Yaskawa INFORM job: DEMO_ROOF_UPPER_0625_3PAINT_17.JBI

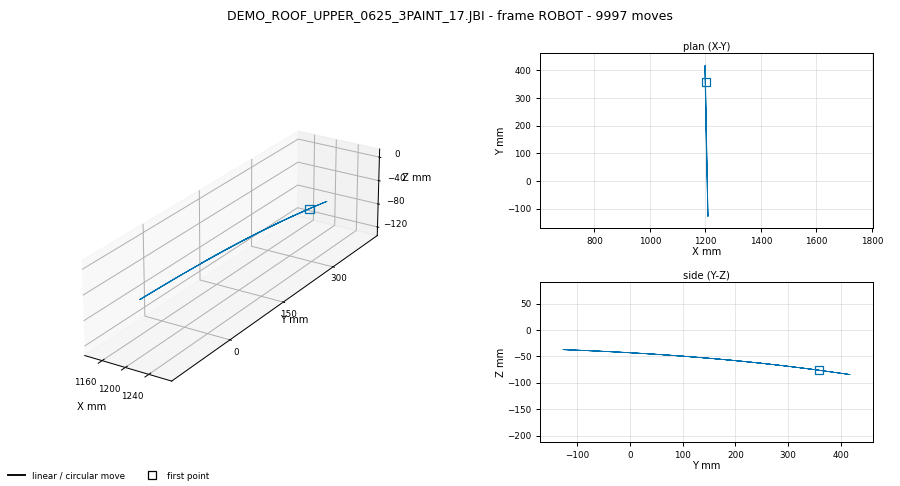
[picture p0: tool path of DEMO_ROOF_UPPER_0625_3PAINT_17.JBI in frame ROBOT, 9997 of 9997 moves have a stored position in this frame; points joined in program order, loops and branches not executed]
/JOB
//NAME DEMO_ROOF_UPPER_0625_3PAINT17
//POS
///NPOS 9997,0,0,0,0,0
///TOOL 0
///USER 0
///POSTYPE ROBOT
///RECTAN
///RCONF 1,0,0,0,0,0,0,0,0,0,0,0,0,0,0,0,0,0,0,0,0,0,0,0
C00000=1200.782,358.357,-76.024,-176.069,8.002,148.413
C00001=1200.786,358.109,-75.991,-176.071,7.999,148.412
C00002=1200.790,357.861,-75.958,-176.072,7.996,148.412
C00003=1200.794,357.613,-75.925,-176.074,7.993,148.412
C00004=1200.798,357.365,-75.891,-176.076,7.989,148.411
C00005=1200.802,357.118,-75.858,-176.078,7.987,148.411
C00006=1200.806,356.870,-75.825,-176.080,7.983,148.411
C00007=1200.811,356.622,-75.792,-176.082,7.980,148.410
C00008=1200.815,356.374,-75.759,-176.083,7.977,148.410
C00009=1200.818,356.127,-75.726,-176.085,7.974,148.410
C00010=1200.822,355.879,-75.693,-176.087,7.971,148.410
C00011=1200.826,355.632,-75.660,-176.089,7.967,148.409
C00012=1200.830,355.384,-75.627,-176.091,7.964,148.409
C00013=1200.835,355.136,-75.594,-176.093,7.962,148.409
C00014=1200.839,354.888,-75.560,-176.094,7.958,148.408
C00015=1200.843,354.641,-75.527,-176.097,7.955,148.408
C00016=1200.847,354.393,-75.494,-176.098,7.952,148.408
C00017=1200.851,354.145,-75.461,-176.101,7.949,148.408
C00018=1200.856,353.897,-75.429,-176.102,7.945,148.407
C00019=1200.860,353.649,-75.395,-176.104,7.943,148.407
C00020=1200.864,353.401,-75.362,-176.106,7.939,148.407
C00021=1200.867,353.154,-75.330,-176.108,7.936,148.406
C00022=1200.871,352.906,-75.297,-176.110,7.933,148.406
C00023=1200.876,352.658,-75.264,-176.112,7.930,148.406
C00024=1200.880,352.410,-75.231,-176.114,7.926,148.406
C00025=1200.884,352.162,-75.198,-176.116,7.924,148.406
C00026=1200.888,351.915,-75.165,-176.118,7.920,148.405
C00027=1200.892,351.667,-75.131,-176.120,7.917,148.405
C00028=1200.896,351.419,-75.100,-176.121,7.914,148.405
C00029=1200.900,351.171,-75.066,-176.124,7.911,148.405
C00030=1200.905,350.924,-75.034,-176.126,7.908,148.404
C00031=1200.909,350.676,-75.001,-176.128,7.905,148.404
C00032=1200.914,350.428,-74.968,-176.129,7.902,148.404
C00033=1200.917,350.181,-74.936,-176.132,7.898,148.404
C00034=1200.921,349.932,-74.903,-176.133,7.896,148.403
C00035=1200.926,349.685,-74.870,-176.135,7.892,148.403
C00036=1200.930,349.437,-74.837,-176.138,7.889,148.403
C00037=1200.934,349.189,-74.804,-176.139,7.887,148.403
C00038=1200.938,348.941,-74.772,-176.142,7.883,148.403
C00039=1200.942,348.693,-74.739,-176.144,7.880,148.402
C00040=1200.946,348.445,-74.706,-176.145,7.877,148.402
C00041=1200.951,348.198,-74.673,-176.147,7.874,148.402
C00042=1200.955,347.950,-74.642,-176.149,7.870,148.401
C00043=1200.959,347.702,-74.608,-176.152,7.867,148.401
C00044=1200.963,347.454,-74.576,-176.153,7.865,148.401
C00045=1200.967,347.206,-74.543,-176.156,7.861,148.401
C00046=1200.971,346.958,-74.511,-176.158,7.858,148.401
C00047=1200.975,346.710,-74.478,-176.159,7.855,148.400
C00048=1200.979,346.463,-74.446,-176.162,7.852,148.400
C00049=1200.984,346.215,-74.413,-176.164,7.849,148.400
C00050=1200.988,345.967,-74.381,-176.166,7.846,148.400
C00051=1200.991,345.720,-74.348,-176.168,7.843,148.400
C00052=1200.996,345.471,-74.316,-176.170,7.840,148.399
C00053=1201.000,345.223,-74.283,-176.172,7.837,148.399
C00054=1201.004,344.975,-74.251,-176.174,7.834,148.399
C00055=1201.008,344.728,-74.218,-176.176,7.830,148.399
C00056=1201.013,344.480,-74.186,-176.178,7.828,148.399
C00057=1201.017,344.232,-74.154,-176.180,7.825,148.398
C00058=1201.021,343.984,-74.121,-176.182,7.821,148.398
C00059=1201.025,343.736,-74.088,-176.184,7.819,148.398
C00060=1201.029,343.489,-74.057,-176.186,7.815,148.398
C00061=1201.034,343.241,-74.023,-176.189,7.812,148.398
C00062=1201.037,342.993,-73.992,-176.191,7.809,148.397
C00063=1201.042,342.745,-73.959,-176.193,7.806,148.397
C00064=1201.046,342.498,-73.927,-176.195,7.803,148.397
C00065=1201.050,342.249,-73.895,-176.197,7.800,148.397
C00066=1201.055,342.001,-73.862,-176.199,7.797,148.397
C00067=1201.058,341.754,-73.830,-176.201,7.794,148.396
C00068=1201.063,341.505,-73.797,-176.203,7.791,148.396
C00069=1201.067,341.258,-73.766,-176.205,7.788,148.396
C00070=1201.071,340.979,-73.729,-176.208,7.784,148.396
C00071=1201.076,340.702,-73.693,-176.210,7.781,148.396
C00072=1201.081,340.422,-73.657,-176.213,7.778,148.396
C00073=1201.086,340.144,-73.620,-176.215,7.774,148.395
C00074=1201.090,339.897,-73.589,-176.217,7.771,148.395
C00075=1201.094,339.649,-73.556,-176.219,7.769,148.395
C00076=1201.098,339.401,-73.524,-176.221,7.765,148.395
C00077=1201.101,339.153,-73.492,-176.224,7.762,148.395
C00078=1201.106,338.905,-73.460,-176.225,7.760,148.395
C00079=1201.110,338.657,-73.428,-176.227,7.756,148.394
C00080=1201.115,338.409,-73.396,-176.230,7.753,148.394
C00081=1201.119,338.161,-73.364,-176.232,7.750,148.394
C00082=1201.123,337.913,-73.332,-176.234,7.747,148.394
C00083=1201.127,337.665,-73.300,-176.236,7.744,148.394
C00084=1201.130,337.418,-73.267,-176.239,7.741,148.394
C00085=1201.136,337.170,-73.235,-176.241,7.738,148.394
C00086=1201.139,336.922,-73.203,-176.243,7.735,148.393
C00087=1201.144,336.673,-73.171,-176.245,7.732,148.393
C00088=1201.148,336.426,-73.140,-176.247,7.730,148.393
C00089=1201.152,336.178,-73.108,-176.249,7.726,148.393
C00090=1201.156,335.930,-73.075,-176.252,7.723,148.393
C00091=1201.160,335.682,-73.044,-176.254,7.720,148.392
C00092=1201.164,335.434,-73.012,-176.256,7.717,148.393
C00093=1201.169,335.186,-72.979,-176.258,7.714,148.392
C00094=1201.173,334.938,-72.949,-176.260,7.711,148.392
C00095=1201.177,334.690,-72.917,-176.263,7.708,148.392
C00096=1201.181,334.442,-72.884,-176.265,7.705,148.392
C00097=1201.186,334.194,-72.853,-176.267,7.702,148.392
C00098=1201.189,333.946,-72.821,-176.269,7.700,148.392
C00099=1201.194,333.699,-72.790,-176.271,7.696,148.392
C00100=1201.198,333.451,-72.757,-176.274,7.693,148.391
C00101=1201.202,333.203,-72.725,-176.276,7.690,148.391
C00102=1201.206,332.955,-72.694,-176.278,7.687,148.391
C00103=1201.210,332.707,-72.663,-176.281,7.684,148.391
C00104=1201.215,332.459,-72.631,-176.283,7.681,148.391
C00105=1201.219,332.211,-72.599,-176.285,7.679,148.391
C00106=1201.223,331.963,-72.567,-176.287,7.676,148.391
C00107=1201.227,331.716,-72.535,-176.289,7.672,148.391
C00108=1201.232,331.467,-72.504,-176.291,7.670,148.390
C00109=1201.236,331.219,-72.472,-176.294,7.667,148.390
C00110=1201.240,330.971,-72.440,-176.296,7.663,148.390
C00111=1201.244,330.724,-72.409,-176.298,7.661,148.390
C00112=1201.248,330.475,-72.378,-176.300,7.658,148.390
C00113=1201.252,330.227,-72.345,-176.303,7.655,148.390
C00114=1201.257,329.980,-72.314,-176.305,7.651,148.390
C00115=1201.261,329.731,-72.283,-176.307,7.649,148.390
C00116=1201.265,329.484,-72.251,-176.310,7.646,148.390
C00117=1201.269,329.235,-72.219,-176.312,7.643,148.389
C00118=1201.273,328.988,-72.189,-176.314,7.640,148.389
C00119=1201.278,328.739,-72.156,-176.316,7.637,148.389
C00120=1201.282,328.492,-72.125,-176.319,7.634,148.389
C00121=1201.286,328.243,-72.094,-176.321,7.631,148.389
C00122=1201.290,327.996,-72.062,-176.323,7.628,148.389
C00123=1201.294,327.747,-72.031,-176.325,7.625,148.389
C00124=1201.299,327.500,-72.000,-176.328,7.622,148.389
C00125=1201.302,327.252,-71.968,-176.330,7.620,148.389
C00126=1201.307,327.004,-71.937,-176.332,7.617,148.389
C00127=1201.311,326.756,-71.905,-176.335,7.613,148.388
C00128=1201.315,326.508,-71.874,-176.337,7.611,148.388
C00129=1201.319,326.260,-71.843,-176.339,7.608,148.388
C00130=1201.324,326.012,-71.812,-176.342,7.605,148.388
C00131=1201.327,325.764,-71.780,-176.343,7.602,148.388
C00132=1201.332,325.516,-71.749,-176.346,7.599,148.388
C00133=1201.336,325.268,-71.717,-176.348,7.596,148.388
C00134=1201.340,325.020,-71.687,-176.351,7.593,148.388
C00135=1201.344,324.772,-71.655,-176.353,7.591,148.388
C00136=1201.349,324.524,-71.624,-176.355,7.587,148.388
C00137=1201.353,324.275,-71.593,-176.358,7.584,148.388
C00138=1201.357,324.028,-71.561,-176.360,7.582,148.388
C00139=1201.361,323.779,-71.530,-176.362,7.579,148.388
C00140=1201.365,323.532,-71.499,-176.365,7.575,148.387
C00141=1201.370,323.284,-71.468,-176.367,7.573,148.387
C00142=1201.374,323.035,-71.437,-176.369,7.570,148.387
C00143=1201.378,322.788,-71.405,-176.372,7.567,148.387
C00144=1201.382,322.539,-71.374,-176.374,7.565,148.387
C00145=1201.387,322.291,-71.343,-176.376,7.561,148.387
C00146=1201.391,322.043,-71.312,-176.379,7.558,148.387
C00147=1201.395,321.795,-71.281,-176.381,7.556,148.387
C00148=1201.400,321.547,-71.250,-176.383,7.553,148.387
C00149=1201.404,321.299,-71.219,-176.386,7.550,148.387
C00150=1201.407,321.052,-71.188,-176.388,7.547,148.387
C00151=1201.412,320.804,-71.157,-176.390,7.544,148.387
C00152=1201.416,320.555,-71.126,-176.393,7.541,148.387
C00153=1201.421,320.307,-71.095,-176.395,7.538,148.387
C00154=1201.424,320.059,-71.064,-176.397,7.536,148.387
C00155=1201.429,319.811,-71.033,-176.400,7.533,148.387
C00156=1201.434,319.563,-71.002,-176.402,7.529,148.386
C00157=1201.437,319.315,-70.971,-176.404,7.527,148.386
C00158=1201.441,319.067,-70.941,-176.407,7.524,148.386
C00159=1201.446,318.819,-70.910,-176.410,7.521,148.386
C00160=1201.450,318.571,-70.878,-176.411,7.518,148.386
C00161=1201.454,318.323,-70.847,-176.414,7.515,148.386
C00162=1201.458,318.075,-70.817,-176.417,7.512,148.386
C00163=1201.462,317.827,-70.786,-176.418,7.510,148.386
C00164=1201.467,317.579,-70.755,-176.421,7.507,148.386
C00165=1201.471,317.331,-70.725,-176.424,7.504,148.386
C00166=1201.475,317.082,-70.694,-176.425,7.501,148.386
C00167=1201.479,316.834,-70.663,-176.428,7.498,148.386
C00168=1201.484,316.586,-70.632,-176.431,7.495,148.386
C00169=1201.488,316.338,-70.601,-176.433,7.492,148.386
C00170=1201.492,316.090,-70.571,-176.435,7.490,148.386
C00171=1201.497,315.842,-70.540,-176.438,7.487,148.386
C00172=1201.501,315.594,-70.510,-176.440,7.484,148.386
C00173=1201.505,315.345,-70.478,-176.443,7.482,148.386
C00174=1201.510,315.070,-70.444,-176.445,7.478,148.386
C00175=1201.515,314.793,-70.411,-176.447,7.475,148.386
C00176=1201.518,314.517,-70.377,-176.450,7.472,148.386
C00177=1201.523,314.241,-70.342,-176.453,7.468,148.386
C00178=1201.528,313.993,-70.312,-176.456,7.466,148.386
C00179=1201.533,313.745,-70.282,-176.458,7.463,148.385
C00180=1201.536,313.496,-70.251,-176.460,7.460,148.385
C00181=1201.541,313.248,-70.220,-176.463,7.458,148.385
C00182=1201.545,313.000,-70.189,-176.465,7.454,148.385
C00183=1201.549,312.753,-70.159,-176.468,7.451,148.386
C00184=1201.554,312.505,-70.129,-176.470,7.449,148.385
C00185=1201.558,312.256,-70.097,-176.472,7.446,148.385
C00186=1201.562,312.008,-70.068,-176.475,7.443,148.385
C00187=1201.567,311.760,-70.037,-176.477,7.441,148.385
C00188=1201.570,311.512,-70.007,-176.480,7.438,148.385
C00189=1201.574,311.264,-69.976,-176.482,7.434,148.385
C00190=1201.579,311.015,-69.946,-176.484,7.432,148.385
C00191=1201.583,310.767,-69.916,-176.487,7.429,148.385
C00192=1201.588,310.520,-69.885,-176.490,7.426,148.385
C00193=1201.592,310.272,-69.855,-176.492,7.424,148.385
C00194=1201.597,310.023,-69.825,-176.494,7.421,148.385
C00195=1201.600,309.775,-69.794,-176.497,7.418,148.385
C00196=1201.605,309.527,-69.763,-176.499,7.415,148.385
C00197=1201.609,309.279,-69.734,-176.501,7.412,148.385
C00198=1201.613,309.031,-69.703,-176.504,7.410,148.385
C00199=1201.617,308.783,-69.673,-176.506,7.407,148.385
C00200=1201.622,308.535,-69.643,-176.509,7.404,148.385
C00201=1201.626,308.287,-69.613,-176.511,7.402,148.385
C00202=1201.630,308.038,-69.582,-176.513,7.399,148.385
C00203=1201.634,307.790,-69.552,-176.516,7.396,148.385
C00204=1201.639,307.542,-69.521,-176.518,7.393,148.385
C00205=1201.643,307.294,-69.492,-176.521,7.390,148.385
C00206=1201.647,307.046,-69.462,-176.523,7.387,148.385
C00207=1201.652,306.798,-69.432,-176.526,7.385,148.385
C00208=1201.656,306.550,-69.402,-176.528,7.382,148.385
C00209=1201.661,306.301,-69.372,-176.531,7.379,148.385
C00210=1201.664,306.054,-69.341,-176.533,7.377,148.385
C00211=1201.669,305.804,-69.311,-176.535,7.374,148.385
C00212=1201.673,305.557,-69.281,-176.538,7.371,148.385
C00213=1201.677,305.308,-69.251,-176.540,7.368,148.385
C00214=1201.681,305.060,-69.221,-176.543,7.365,148.385
C00215=1201.686,304.812,-69.191,-176.545,7.363,148.385
C00216=1201.689,304.565,-69.161,-176.548,7.360,148.385
C00217=1201.694,304.316,-69.131,-176.550,7.357,148.385
C00218=1201.699,304.068,-69.101,-176.553,7.355,148.385
C00219=1201.703,303.820,-69.071,-176.555,7.352,148.385
C00220=1201.707,303.572,-69.041,-176.558,7.349,148.385
C00221=1201.711,303.324,-69.011,-176.560,7.347,148.386
C00222=1201.716,303.075,-68.981,-176.563,7.344,148.386
C00223=1201.720,302.827,-68.952,-176.565,7.341,148.386
C00224=1201.724,302.579,-68.921,-176.567,7.338,148.385
C00225=1201.728,302.331,-68.892,-176.570,7.335,148.385
C00226=1201.733,302.083,-68.862,-176.572,7.333,148.385
C00227=1201.738,301.834,-68.832,-176.575,7.330,148.385
C00228=1201.741,301.587,-68.802,-176.577,7.327,148.385
C00229=1201.746,301.338,-68.773,-176.579,7.325,148.386
C00230=1201.750,301.090,-68.743,-176.582,7.322,148.386
C00231=1201.754,300.842,-68.713,-176.584,7.319,148.386
C00232=1201.759,300.594,-68.683,-176.587,7.316,148.386
C00233=1201.763,300.346,-68.654,-176.590,7.313,148.386
C00234=1201.768,300.097,-68.624,-176.592,7.311,148.386
C00235=1201.772,299.849,-68.594,-176.594,7.308,148.386
C00236=1201.776,299.601,-68.564,-176.597,7.305,148.386
C00237=1201.780,299.353,-68.535,-176.599,7.303,148.386
C00238=1201.784,299.105,-68.505,-176.602,7.300,148.386
C00239=1201.789,298.856,-68.475,-176.604,7.298,148.386
C00240=1201.793,298.608,-68.446,-176.607,7.295,148.386
C00241=1201.797,298.359,-68.416,-176.610,7.292,148.386
C00242=1201.802,298.111,-68.387,-176.612,7.290,148.386
C00243=1201.805,297.864,-68.357,-176.614,7.287,148.386
C00244=1201.810,297.615,-68.327,-176.616,7.284,148.386
C00245=1201.814,297.367,-68.298,-176.619,7.281,148.386
C00246=1201.819,297.118,-68.268,-176.622,7.278,148.386
C00247=1201.823,296.870,-68.238,-176.624,7.276,148.386
C00248=1201.827,296.622,-68.209,-176.627,7.273,148.386
C00249=1201.832,296.374,-68.180,-176.629,7.271,148.386
C00250=1201.836,296.126,-68.150,-176.632,7.268,148.386
C00251=1201.840,295.878,-68.121,-176.635,7.265,148.387
C00252=1201.844,295.630,-68.091,-176.637,7.263,148.387
C00253=1201.849,295.381,-68.062,-176.640,7.260,148.387
C00254=1201.853,295.133,-68.032,-176.642,7.258,148.387
C00255=1201.857,294.885,-68.003,-176.644,7.255,148.387
C00256=1201.861,294.636,-67.973,-176.647,7.252,148.387
C00257=1201.865,294.388,-67.944,-176.649,7.250,148.387
C00258=1201.870,294.141,-67.915,-176.652,7.247,148.387
C00259=1201.875,293.892,-67.886,-176.654,7.244,148.387
C00260=1201.879,293.643,-67.857,-176.657,7.241,148.387
C00261=1201.883,293.395,-67.827,-176.659,7.238,148.387
C00262=1201.887,293.147,-67.798,-176.662,7.236,148.387
C00263=1201.891,292.899,-67.768,-176.664,7.233,148.387
C00264=1201.895,292.650,-67.739,-176.666,7.231,148.387
C00265=1201.900,292.403,-67.710,-176.670,7.228,148.387
C00266=1201.905,292.154,-67.681,-176.672,7.226,148.387
C00267=1201.909,291.906,-67.652,-176.674,7.223,148.387
C00268=1201.913,291.657,-67.622,-176.677,7.220,148.387
C00269=1201.917,291.409,-67.593,-176.679,7.218,148.387
C00270=1201.922,291.162,-67.564,-176.682,7.215,148.388
C00271=1201.927,290.913,-67.535,-176.684,7.213,148.388
C00272=1201.931,290.664,-67.505,-176.687,7.210,148.388
C00273=1201.935,290.416,-67.476,-176.689,7.207,148.388
C00274=1201.939,290.168,-67.448,-176.692,7.204,148.388
C00275=1201.943,289.920,-67.419,-176.695,7.202,148.388
C00276=1201.948,289.672,-67.389,-176.697,7.199,148.388
C00277=1201.952,289.423,-67.360,-176.700,7.196,148.388
C00278=1201.957,289.149,-67.328,-176.702,7.193,148.388
C00279=1201.962,288.874,-67.296,-176.705,7.190,148.388
C00280=1201.966,288.599,-67.264,-176.708,7.189,148.388
C00281=1201.971,288.326,-67.232,-176.710,7.186,148.388
C00282=1201.976,288.077,-67.203,-176.713,7.183,148.388
C00283=1201.980,287.829,-67.174,-176.715,7.180,148.388
C00284=1201.984,287.581,-67.144,-176.718,7.177,148.388
C00285=1201.988,287.332,-67.116,-176.720,7.174,148.389
C00286=1201.993,287.085,-67.087,-176.723,7.172,148.389
C00287=1201.997,286.836,-67.058,-176.726,7.169,148.389
C00288=1202.002,286.588,-67.029,-176.728,7.167,148.389
C00289=1202.005,286.339,-67.001,-176.731,7.164,148.389
C00290=1202.010,286.091,-66.972,-176.733,7.162,148.389
C00291=1202.015,285.843,-66.943,-176.735,7.159,148.389
C00292=1202.019,285.594,-66.913,-176.738,7.157,148.389
C00293=1202.023,285.346,-66.886,-176.741,7.154,148.389
C00294=1202.027,285.098,-66.856,-176.743,7.152,148.389
C00295=1202.032,284.849,-66.827,-176.746,7.149,148.389
C00296=1202.037,284.602,-66.798,-176.748,7.146,148.389
C00297=1202.040,284.353,-66.770,-176.751,7.144,148.390
C00298=1202.044,284.105,-66.741,-176.754,7.141,148.390
C00299=1202.050,283.857,-66.712,-176.756,7.139,148.390
C00300=1202.053,283.608,-66.684,-176.758,7.136,148.390
C00301=1202.057,283.360,-66.655,-176.761,7.134,148.390
C00302=1202.063,283.112,-66.626,-176.764,7.131,148.390
C00303=1202.066,282.863,-66.598,-176.766,7.129,148.390
C00304=1202.070,282.615,-66.569,-176.769,7.126,148.390
C00305=1202.076,282.367,-66.540,-176.771,7.124,148.390
C00306=1202.079,282.118,-66.512,-176.773,7.121,148.390
C00307=1202.084,281.870,-66.483,-176.776,7.119,148.391
C00308=1202.089,281.622,-66.455,-176.779,7.116,148.391
C00309=1202.092,281.373,-66.426,-176.781,7.113,148.391
C00310=1202.097,281.125,-66.397,-176.784,7.110,148.391
C00311=1202.102,280.877,-66.369,-176.786,7.108,148.391
C00312=1202.105,280.628,-66.340,-176.789,7.106,148.391
C00313=1202.110,280.380,-66.312,-176.791,7.103,148.391
C00314=1202.114,280.131,-66.284,-176.794,7.100,148.391
C00315=1202.119,279.884,-66.255,-176.796,7.098,148.391
C00316=1202.123,279.635,-66.227,-176.799,7.096,148.392
C00317=1202.127,279.386,-66.198,-176.801,7.093,148.392
C00318=1202.132,279.138,-66.170,-176.804,7.090,148.392
C00319=1202.136,278.889,-66.141,-176.806,7.088,148.392
C00320=1202.140,278.642,-66.113,-176.809,7.085,148.392
C00321=1202.145,278.393,-66.084,-176.811,7.083,148.392
C00322=1202.149,278.145,-66.056,-176.814,7.080,148.392
C00323=1202.153,277.897,-66.028,-176.816,7.078,148.392
C00324=1202.157,277.648,-66.000,-176.819,7.075,148.392
C00325=1202.162,277.400,-65.971,-176.821,7.073,148.393
C00326=1202.166,277.151,-65.943,-176.824,7.070,148.393
C00327=1202.171,276.903,-65.915,-176.826,7.068,148.393
C00328=1202.175,276.654,-65.886,-176.830,7.065,148.393
C00329=1202.180,276.406,-65.858,-176.832,7.063,148.393
C00330=1202.184,276.158,-65.830,-176.834,7.060,148.393
C00331=1202.189,275.909,-65.802,-176.837,7.058,148.393
C00332=1202.193,275.661,-65.773,-176.840,7.055,148.393
C00333=1202.198,275.413,-65.745,-176.842,7.053,148.393
C00334=1202.201,275.164,-65.717,-176.845,7.050,148.393
C00335=1202.206,274.916,-65.689,-176.847,7.048,148.394
C00336=1202.210,274.667,-65.660,-176.850,7.045,148.394
C00337=1202.215,274.419,-65.633,-176.852,7.043,148.394
C00338=1202.219,274.171,-65.604,-176.855,7.041,148.394
C00339=1202.223,273.923,-65.576,-176.857,7.038,148.394
C00340=1202.227,273.674,-65.548,-176.859,7.036,148.394
C00341=1202.232,273.426,-65.520,-176.862,7.033,148.394
C00342=1202.236,273.177,-65.491,-176.865,7.031,148.395
C00343=1202.240,272.930,-65.464,-176.867,7.028,148.395
C00344=1202.246,272.681,-65.436,-176.870,7.026,148.395
C00345=1202.249,272.432,-65.408,-176.873,7.023,148.395
C00346=1202.254,272.184,-65.380,-176.875,7.021,148.395
C00347=1202.258,271.935,-65.351,-176.878,7.018,148.395
C00348=1202.263,271.687,-65.324,-176.880,7.016,148.395
C00349=1202.266,271.439,-65.295,-176.882,7.014,148.395
C00350=1202.271,271.190,-65.268,-176.885,7.011,148.395
C00351=1202.276,270.942,-65.240,-176.888,7.009,148.396
C00352=1202.280,270.694,-65.212,-176.890,7.006,148.396
C00353=1202.284,270.446,-65.184,-176.893,7.004,148.396
C00354=1202.289,270.196,-65.156,-176.896,7.001,148.396
C00355=1202.293,269.948,-65.128,-176.898,6.999,148.396
C00356=1202.297,269.700,-65.100,-176.901,6.996,148.396
C00357=1202.302,269.451,-65.073,-176.903,6.994,148.397
C00358=1202.307,269.203,-65.045,-176.905,6.992,148.397
C00359=1202.311,268.955,-65.017,-176.908,6.989,148.397
C00360=1202.315,268.706,-64.990,-176.911,6.987,148.397
C00361=1202.320,268.458,-64.962,-176.913,6.984,148.397
C00362=1202.323,268.210,-64.934,-176.915,6.982,148.397
C00363=1202.329,267.961,-64.906,-176.919,6.979,148.397
C00364=1202.333,267.713,-64.878,-176.921,6.977,148.397
C00365=1202.337,267.464,-64.850,-176.923,6.975,148.398
C00366=1202.342,267.216,-64.823,-176.926,6.972,148.398
C00367=1202.346,266.968,-64.795,-176.928,6.970,148.398
C00368=1202.350,266.719,-64.768,-176.931,6.967,148.398
C00369=1202.355,266.471,-64.739,-176.934,6.965,148.398
C00370=1202.360,266.222,-64.712,-176.936,6.962,148.398
C00371=1202.363,265.974,-64.684,-176.939,6.960,148.399
C00372=1202.368,265.725,-64.657,-176.941,6.958,148.399
C00373=1202.372,265.477,-64.629,-176.944,6.955,148.399
C00374=1202.377,265.228,-64.602,-176.946,6.953,148.399
C00375=1202.381,264.980,-64.574,-176.949,6.950,148.399
C00376=1202.386,264.732,-64.547,-176.952,6.948,148.399
C00377=1202.389,264.483,-64.519,-176.954,6.946,148.399
C00378=1202.394,264.235,-64.492,-176.957,6.943,148.399
C00379=1202.399,263.986,-64.464,-176.959,6.941,148.400
C00380=1202.404,263.738,-64.436,-176.962,6.938,148.400
C00381=1202.407,263.489,-64.408,-176.964,6.936,148.400
C00382=1202.412,263.217,-64.379,-176.967,6.933,148.400
C00383=1202.418,262.944,-64.349,-176.970,6.932,148.400
C00384=1202.422,262.670,-64.318,-176.973,6.929,148.400
C00385=1202.427,262.398,-64.289,-176.976,6.926,148.401
C00386=1202.431,262.150,-64.261,-176.978,6.924,148.401
C00387=1202.436,261.902,-64.234,-176.981,6.921,148.401
C00388=1202.440,261.652,-64.206,-176.983,6.919,148.401
C00389=1202.444,261.405,-64.179,-176.985,6.917,148.401
C00390=1202.449,261.156,-64.152,-176.989,6.914,148.402
C00391=1202.453,260.908,-64.124,-176.991,6.912,148.402
C00392=1202.458,260.658,-64.097,-176.993,6.910,148.402
C00393=1202.462,260.411,-64.069,-176.996,6.907,148.402
C00394=1202.467,260.162,-64.042,-176.999,6.905,148.402
C00395=1202.471,259.914,-64.015,-177.001,6.902,148.402
C00396=1202.476,259.665,-63.988,-177.003,6.900,148.402
C00397=1202.480,259.416,-63.960,-177.006,6.898,148.403
C00398=1202.484,259.168,-63.933,-177.009,6.895,148.403
C00399=1202.488,258.920,-63.906,-177.011,6.893,148.403
C00400=1202.493,258.671,-63.879,-177.014,6.891,148.403
C00401=1202.497,258.423,-63.852,-177.017,6.888,148.403
C00402=1202.501,258.174,-63.824,-177.019,6.886,148.403
C00403=1202.506,257.926,-63.797,-177.022,6.884,148.404
C00404=1202.511,257.677,-63.770,-177.024,6.881,148.404
C00405=1202.515,257.429,-63.743,-177.027,6.879,148.404
C00406=1202.520,257.180,-63.716,-177.029,6.877,148.404
C00407=1202.524,256.932,-63.689,-177.032,6.874,148.404
C00408=1202.528,256.684,-63.662,-177.034,6.872,148.405
C00409=1202.532,256.434,-63.635,-177.037,6.869,148.405
C00410=1202.537,256.186,-63.608,-177.040,6.867,148.405
C00411=1202.542,255.937,-63.581,-177.042,6.865,148.405
C00412=1202.546,255.689,-63.554,-177.045,6.863,148.405
C00413=1202.550,255.441,-63.527,-177.047,6.860,148.405
C00414=1202.555,255.192,-63.500,-177.050,6.859,148.406
C00415=1202.560,254.944,-63.473,-177.052,6.856,148.406
C00416=1202.564,254.695,-63.446,-177.055,6.854,148.406
C00417=1202.568,254.446,-63.419,-177.057,6.852,148.406
C00418=1202.572,254.198,-63.392,-177.060,6.849,148.406
C00419=1202.577,253.949,-63.365,-177.063,6.847,148.407
C00420=1202.582,253.701,-63.338,-177.065,6.845,148.407
C00421=1202.586,253.453,-63.312,-177.067,6.843,148.407
C00422=1202.590,253.204,-63.285,-177.071,6.840,148.407
C00423=1202.595,252.956,-63.257,-177.073,6.838,148.407
C00424=1202.599,252.707,-63.231,-177.075,6.836,148.408
C00425=1202.603,252.459,-63.204,-177.078,6.833,148.408
C00426=1202.608,252.211,-63.177,-177.081,6.831,148.408
C00427=1202.613,251.962,-63.150,-177.083,6.829,148.408
C00428=1202.617,251.713,-63.124,-177.086,6.826,148.408
C00429=1202.622,251.465,-63.097,-177.088,6.824,148.408
C00430=1202.626,251.216,-63.070,-177.091,6.822,148.409
C00431=1202.630,250.968,-63.043,-177.093,6.819,148.409
C00432=1202.634,250.719,-63.016,-177.096,6.817,148.409
C00433=1202.638,250.471,-62.990,-177.098,6.815,148.409
C00434=1202.643,250.222,-62.963,-177.101,6.813,148.409
C00435=1202.648,249.973,-62.936,-177.104,6.810,148.410
C00436=1202.652,249.725,-62.910,-177.106,6.808,148.410
C00437=1202.656,249.476,-62.883,-177.108,6.806,148.410
C00438=1202.661,249.227,-62.856,-177.112,6.804,148.410
C00439=1202.665,248.979,-62.830,-177.114,6.801,148.410
C00440=1202.670,248.731,-62.803,-177.116,6.800,148.411
C00441=1202.674,248.482,-62.777,-177.119,6.797,148.411
C00442=1202.679,248.233,-62.750,-177.122,6.795,148.411
C00443=1202.683,247.985,-62.724,-177.124,6.793,148.411
C00444=1202.688,247.736,-62.697,-177.126,6.791,148.411
C00445=1202.693,247.488,-62.670,-177.130,6.788,148.412
C00446=1202.697,247.240,-62.644,-177.132,6.786,148.412
C00447=1202.702,246.991,-62.618,-177.134,6.784,148.412
C00448=1202.706,246.743,-62.591,-177.137,6.781,148.412
C00449=1202.710,246.494,-62.564,-177.140,6.779,148.412
C00450=1202.715,246.245,-62.538,-177.142,6.777,148.413
C00451=1202.719,245.997,-62.511,-177.145,6.775,148.413
C00452=1202.723,245.748,-62.486,-177.148,6.772,148.413
C00453=1202.728,245.500,-62.458,-177.150,6.770,148.413
C00454=1202.732,245.251,-62.433,-177.152,6.768,148.414
C00455=1202.737,245.002,-62.406,-177.155,6.766,148.414
C00456=1202.741,244.753,-62.380,-177.158,6.764,148.414
C00457=1202.745,244.505,-62.353,-177.160,6.761,148.414
C00458=1202.750,244.257,-62.326,-177.163,6.760,148.414
C00459=1202.754,244.008,-62.301,-177.165,6.758,148.415
C00460=1202.760,243.760,-62.275,-177.168,6.755,148.415
C00461=1202.764,243.511,-62.248,-177.171,6.753,148.415
C00462=1202.768,243.262,-62.222,-177.173,6.751,148.415
C00463=1202.772,243.014,-62.195,-177.175,6.749,148.415
C00464=1202.777,242.765,-62.170,-177.178,6.746,148.415
C00465=1202.781,242.517,-62.143,-177.181,6.744,148.416
C00466=1202.786,242.268,-62.117,-177.183,6.742,148.416
C00467=1202.790,242.019,-62.090,-177.185,6.740,148.416
C00468=1202.794,241.771,-62.064,-177.189,6.737,148.416
C00469=1202.799,241.523,-62.039,-177.191,6.735,148.417
C00470=1202.804,241.274,-62.012,-177.193,6.733,148.417
C00471=1202.808,241.025,-61.986,-177.196,6.731,148.417
C00472=1202.812,240.776,-61.960,-177.199,6.728,148.417
C00473=1202.817,240.528,-61.933,-177.201,6.727,148.418
C00474=1202.821,240.279,-61.907,-177.204,6.724,148.418
C00475=1202.826,240.031,-61.882,-177.206,6.723,148.418
C00476=1202.831,239.783,-61.855,-177.209,6.720,148.418
C00477=1202.835,239.534,-61.829,-177.212,6.718,148.418
C00478=1202.839,239.285,-61.803,-177.214,6.716,148.419
C00479=1202.844,239.036,-61.777,-177.217,6.714,148.419
C00480=1202.849,238.788,-61.751,-177.219,6.712,148.419
C00481=1202.853,238.540,-61.725,-177.222,6.709,148.419
C00482=1202.857,238.291,-61.699,-177.224,6.707,148.419
C00483=1202.862,238.042,-61.673,-177.227,6.705,148.420
C00484=1202.866,237.793,-61.647,-177.230,6.703,148.420
C00485=1202.871,237.545,-61.621,-177.232,6.700,148.420
C00486=1202.875,237.273,-61.593,-177.235,6.699,148.421
C00487=1202.880,237.002,-61.565,-177.238,6.696,148.421
C00488=1202.886,236.731,-61.536,-177.241,6.694,148.421
C00489=1202.891,236.459,-61.508,-177.244,6.691,148.421
C00490=1202.895,236.210,-61.482,-177.246,6.689,148.421
C00491=1202.899,235.961,-61.457,-177.249,6.687,148.422
C00492=1202.904,235.714,-61.430,-177.251,6.685,148.422
C00493=1202.908,235.465,-61.405,-177.254,6.683,148.422
C00494=1202.913,235.216,-61.378,-177.257,6.681,148.423
C00495=1202.917,234.967,-61.353,-177.259,6.679,148.423
C00496=1202.922,234.719,-61.327,-177.262,6.677,148.423
C00497=1202.926,234.470,-61.301,-177.264,6.675,148.423
C00498=1202.930,234.221,-61.276,-177.266,6.673,148.423
C00499=1202.935,233.973,-61.250,-177.270,6.670,148.424
C00500=1202.939,233.724,-61.225,-177.272,6.668,148.424
C00501=1202.944,233.475,-61.198,-177.274,6.666,148.424
C00502=1202.948,233.226,-61.172,-177.277,6.664,148.424
C00503=1202.953,232.978,-61.147,-177.280,6.662,148.425
C00504=1202.958,232.730,-61.121,-177.282,6.659,148.425
C00505=1202.962,232.481,-61.096,-177.285,6.657,148.425
C00506=1202.967,232.233,-61.070,-177.288,6.656,148.425
C00507=1202.971,231.984,-61.044,-177.290,6.653,148.426
C00508=1202.975,231.735,-61.019,-177.292,6.652,148.426
C00509=1202.980,231.486,-60.994,-177.295,6.650,148.426
C00510=1202.984,231.237,-60.968,-177.298,6.647,148.426
C00511=1202.989,230.989,-60.943,-177.300,6.645,148.427
C00512=1202.993,230.741,-60.917,-177.303,6.643,148.427
C00513=1202.998,230.492,-60.891,-177.306,6.641,148.427
C00514=1203.002,230.243,-60.866,-177.308,6.639,148.427
C00515=1203.007,229.995,-60.840,-177.310,6.637,148.428
C00516=1203.011,229.746,-60.815,-177.314,6.635,148.428
C00517=1203.015,229.497,-60.789,-177.316,6.632,148.428
C00518=1203.020,229.249,-60.764,-177.318,6.631,148.428
C00519=1203.025,229.000,-60.738,-177.321,6.629,148.429
C00520=1203.029,228.752,-60.713,-177.324,6.627,148.429
C00521=1203.034,228.502,-60.688,-177.326,6.625,148.429
C00522=1203.038,228.253,-60.662,-177.329,6.622,148.429
C00523=1203.043,228.005,-60.637,-177.332,6.620,148.430
C00524=1203.047,227.756,-60.611,-177.334,6.618,148.430
C00525=1203.052,227.508,-60.586,-177.336,6.616,148.430
C00526=1203.057,227.259,-60.561,-177.339,6.614,148.430
C00527=1203.061,227.010,-60.535,-177.342,6.613,148.431
C00528=1203.066,226.762,-60.509,-177.344,6.610,148.431
C00529=1203.070,226.513,-60.484,-177.347,6.608,148.431
C00530=1203.075,226.264,-60.459,-177.350,6.606,148.432
C00531=1203.078,226.016,-60.434,-177.352,6.604,148.432
C00532=1203.084,225.767,-60.409,-177.355,6.602,148.432
C00533=1203.088,225.518,-60.383,-177.357,6.600,148.432
C00534=1203.092,225.269,-60.358,-177.360,6.598,148.433
C00535=1203.097,225.021,-60.333,-177.363,6.596,148.433
C00536=1203.101,224.772,-60.307,-177.365,6.593,148.433
C00537=1203.106,224.523,-60.283,-177.368,6.592,148.433
C00538=1203.110,224.275,-60.257,-177.370,6.590,148.434
C00539=1203.115,224.026,-60.233,-177.373,6.588,148.434
C00540=1203.119,223.777,-60.207,-177.375,6.586,148.434
C00541=1203.124,223.529,-60.182,-177.378,6.584,148.434
C00542=1203.129,223.280,-60.157,-177.381,6.581,148.435
C00543=1203.134,223.032,-60.131,-177.384,6.579,148.435
C00544=1203.137,222.783,-60.107,-177.386,6.577,148.435
C00545=1203.142,222.535,-60.081,-177.389,6.575,148.436
C00546=1203.147,222.285,-60.056,-177.391,6.574,148.436
C00547=1203.152,222.036,-60.032,-177.394,6.572,148.436
C00548=1203.155,221.788,-60.007,-177.396,6.570,148.436
C00549=1203.160,221.539,-59.982,-177.399,6.568,148.437
C00550=1203.165,221.290,-59.956,-177.402,6.565,148.437
C00551=1203.170,221.042,-59.931,-177.404,6.563,148.437
C00552=1203.173,220.793,-59.906,-177.407,6.561,148.438
C00553=1203.178,220.544,-59.882,-177.409,6.559,148.438
C00554=1203.183,220.295,-59.857,-177.412,6.557,148.438
C00555=1203.187,220.047,-59.832,-177.415,6.556,148.438
C00556=1203.192,219.798,-59.807,-177.417,6.554,148.439
C00557=1203.196,219.550,-59.781,-177.419,6.552,148.439
C00558=1203.201,219.301,-59.757,-177.423,6.549,148.439
C00559=1203.205,219.052,-59.732,-177.425,6.547,148.439
C00560=1203.210,218.804,-59.707,-177.428,6.545,148.440
C00561=1203.215,218.554,-59.682,-177.430,6.543,148.440
C00562=1203.219,218.306,-59.658,-177.433,6.541,148.440
C00563=1203.223,218.057,-59.632,-177.435,6.539,148.441
C00564=1203.228,217.809,-59.608,-177.438,6.538,148.441
C00565=1203.233,217.560,-59.583,-177.441,6.536,148.441
C00566=1203.237,217.311,-59.558,-177.443,6.534,148.442
C00567=1203.241,217.063,-59.534,-177.446,6.531,148.442
C00568=1203.246,216.813,-59.508,-177.449,6.529,148.442
C00569=1203.251,216.565,-59.484,-177.451,6.527,148.442
C00570=1203.255,216.316,-59.460,-177.454,6.525,148.443
C00571=1203.260,216.067,-59.435,-177.456,6.524,148.443
C00572=1203.264,215.819,-59.410,-177.459,6.522,148.443
C00573=1203.269,215.570,-59.385,-177.461,6.520,148.443
C00574=1203.273,215.321,-59.361,-177.464,6.518,148.444
C00575=1203.278,215.072,-59.336,-177.467,6.516,148.444
C00576=1203.282,214.823,-59.312,-177.469,6.514,148.444
C00577=1203.287,214.575,-59.287,-177.472,6.511,148.445
C00578=1203.292,214.326,-59.262,-177.475,6.510,148.445
C00579=1203.296,214.077,-59.237,-177.477,6.507,148.445
C00580=1203.301,213.829,-59.213,-177.480,6.506,148.445
C00581=1203.305,213.580,-59.188,-177.483,6.504,148.446
C00582=1203.310,213.331,-59.163,-177.485,6.502,148.446
C00583=1203.314,213.082,-59.139,-177.488,6.500,148.446
C00584=1203.319,212.834,-59.115,-177.490,6.498,148.447
C00585=1203.323,212.585,-59.090,-177.493,6.496,148.447
C00586=1203.328,212.336,-59.066,-177.495,6.494,148.447
C00587=1203.333,212.087,-59.041,-177.498,6.492,148.448
C00588=1203.337,211.839,-59.017,-177.501,6.491,148.448
C00589=1203.341,211.590,-58.992,-177.503,6.489,148.448
C00590=1203.347,211.319,-58.966,-177.506,6.486,148.449
C00591=1203.352,211.049,-58.939,-177.509,6.484,148.449
C00592=1203.356,210.779,-58.913,-177.512,6.483,148.449
C00593=1203.361,210.508,-58.886,-177.515,6.480,148.450
C00594=1203.366,210.259,-58.862,-177.518,6.478,148.450
C00595=1203.371,210.011,-58.838,-177.520,6.476,148.450
C00596=1203.375,209.762,-58.814,-177.523,6.474,148.451
C00597=1203.380,209.513,-58.789,-177.526,6.473,148.451
C00598=1203.384,209.265,-58.765,-177.528,6.470,148.451
C00599=1203.389,209.016,-58.740,-177.530,6.469,148.451
C00600=1203.393,208.767,-58.716,-177.533,6.467,148.452
C00601=1203.398,208.518,-58.692,-177.536,6.465,148.452
C00602=1203.403,208.269,-58.667,-177.538,6.463,148.452
C00603=1203.407,208.020,-58.643,-177.541,6.461,148.453
C00604=1203.411,207.772,-58.619,-177.544,6.459,148.453
C00605=1203.416,207.523,-58.594,-177.546,6.458,148.453
C00606=1203.420,207.274,-58.570,-177.549,6.455,148.453
C00607=1203.425,207.025,-58.547,-177.552,6.453,148.454
C00608=1203.430,206.776,-58.522,-177.554,6.451,148.454
C00609=1203.435,206.528,-58.498,-177.557,6.449,148.454
C00610=1203.438,206.279,-58.474,-177.560,6.447,148.455
C00611=1203.444,206.030,-58.450,-177.562,6.446,148.455
C00612=1203.448,205.781,-58.426,-177.565,6.444,148.455
C00613=1203.453,205.533,-58.401,-177.567,6.442,148.456
C00614=1203.457,205.284,-58.377,-177.570,6.440,148.456
C00615=1203.462,205.034,-58.353,-177.572,6.438,148.456
C00616=1203.466,204.786,-58.329,-177.575,6.436,148.457
C00617=1203.471,204.538,-58.305,-177.578,6.434,148.457
C00618=1203.475,204.288,-58.282,-177.580,6.432,148.457
C00619=1203.480,204.040,-58.257,-177.583,6.431,148.458
C00620=1203.485,203.791,-58.233,-177.586,6.429,148.458
C00621=1203.490,203.542,-58.209,-177.588,6.427,148.458
C00622=1203.493,203.293,-58.185,-177.591,6.425,148.459
C00623=1203.498,203.045,-58.161,-177.593,6.423,148.459
C00624=1203.503,202.795,-58.137,-177.596,6.421,148.459
C00625=1203.508,202.547,-58.113,-177.599,6.420,148.460
C00626=1203.512,202.298,-58.090,-177.601,6.418,148.460
C00627=1203.517,202.050,-58.066,-177.604,6.416,148.460
C00628=1203.521,201.801,-58.041,-177.606,6.414,148.461
C00629=1203.525,201.551,-58.018,-177.609,6.412,148.461
C00630=1203.530,201.303,-57.994,-177.612,6.410,148.461
C00631=1203.535,201.054,-57.970,-177.614,6.408,148.462
C00632=1203.539,200.805,-57.946,-177.617,6.407,148.462
C00633=1203.544,200.556,-57.922,-177.619,6.405,148.462
C00634=1203.548,200.308,-57.898,-177.622,6.403,148.463
C00635=1203.553,200.059,-57.875,-177.625,6.401,148.463
C00636=1203.558,199.810,-57.851,-177.627,6.399,148.463
C00637=1203.562,199.561,-57.827,-177.630,6.397,148.464
C00638=1203.567,199.313,-57.803,-177.633,6.396,148.464
C00639=1203.571,199.064,-57.780,-177.635,6.394,148.464
C00640=1203.576,198.815,-57.757,-177.638,6.392,148.465
C00641=1203.581,198.565,-57.732,-177.641,6.390,148.465
C00642=1203.585,198.316,-57.708,-177.643,6.388,148.465
C00643=1203.590,198.068,-57.684,-177.646,6.386,148.465
C00644=1203.594,197.819,-57.661,-177.648,6.384,148.466
C00645=1203.599,197.570,-57.637,-177.651,6.383,148.466
C00646=1203.604,197.322,-57.613,-177.653,6.381,148.466
C00647=1203.608,197.072,-57.590,-177.656,6.379,148.467
C00648=1203.613,196.823,-57.567,-177.659,6.377,148.467
C00649=1203.617,196.575,-57.543,-177.661,6.375,148.468
C00650=1203.622,196.326,-57.519,-177.664,6.373,148.468
C00651=1203.627,196.077,-57.496,-177.667,6.372,148.468
C00652=1203.631,195.829,-57.472,-177.669,6.370,148.469
C00653=1203.636,195.580,-57.448,-177.672,6.368,148.469
C00654=1203.640,195.331,-57.425,-177.675,6.366,148.469
C00655=1203.645,195.081,-57.402,-177.677,6.364,148.470
C00656=1203.650,194.833,-57.378,-177.680,6.363,148.470
C00657=1203.654,194.584,-57.354,-177.682,6.362,148.470
C00658=1203.658,194.335,-57.331,-177.685,6.360,148.471
C00659=1203.663,194.086,-57.308,-177.687,6.358,148.471
C00660=1203.667,193.838,-57.284,-177.690,6.356,148.471
C00661=1203.672,193.589,-57.261,-177.693,6.354,148.472
C00662=1203.677,193.340,-57.237,-177.695,6.352,148.472
C00663=1203.681,193.091,-57.214,-177.698,6.351,148.472
C00664=1203.687,192.842,-57.191,-177.701,6.349,148.473
C00665=1203.691,192.594,-57.167,-177.703,6.347,148.473
C00666=1203.696,192.345,-57.144,-177.706,6.345,148.473
C00667=1203.701,192.096,-57.120,-177.709,6.343,148.474
C00668=1203.704,191.847,-57.097,-177.711,6.342,148.474
C00669=1203.709,191.598,-57.074,-177.714,6.340,148.475
C00670=1203.714,191.349,-57.051,-177.717,6.338,148.475
C00671=1203.719,191.100,-57.027,-177.719,6.336,148.475
C00672=1203.723,190.851,-57.004,-177.722,6.334,148.476
C00673=1203.728,190.602,-56.981,-177.725,6.332,148.476
C00674=1203.733,190.353,-56.957,-177.727,6.331,148.476
C00675=1203.737,190.104,-56.934,-177.729,6.330,148.477
C00676=1203.742,189.856,-56.912,-177.732,6.328,148.477
C00677=1203.747,189.607,-56.888,-177.735,6.326,148.477
C00678=1203.751,189.359,-56.864,-177.737,6.324,148.478
C00679=1203.756,189.110,-56.841,-177.740,6.322,148.478
C00680=1203.760,188.860,-56.819,-177.743,6.321,148.478
C00681=1203.765,188.611,-56.795,-177.745,6.319,148.479
C00682=1203.769,188.362,-56.772,-177.748,6.317,148.479
C00683=1203.774,188.113,-56.749,-177.751,6.315,148.479
C00684=1203.779,187.865,-56.726,-177.753,6.313,148.480
C00685=1203.783,187.616,-56.703,-177.756,6.312,148.480
C00686=1203.788,187.367,-56.679,-177.758,6.311,148.481
C00687=1203.793,187.118,-56.656,-177.761,6.309,148.481
C00688=1203.797,186.869,-56.633,-177.763,6.307,148.481
C00689=1203.801,186.620,-56.610,-177.766,6.305,148.482
C00690=1203.806,186.371,-56.587,-177.769,6.303,148.482
C00691=1203.811,186.123,-56.564,-177.771,6.301,148.482
C00692=1203.815,185.874,-56.541,-177.774,6.300,148.483
C00693=1203.820,185.624,-56.518,-177.777,6.298,148.483
C00694=1203.825,185.356,-56.493,-177.779,6.296,148.483
C00695=1203.830,185.086,-56.468,-177.782,6.294,148.484
C00696=1203.835,184.816,-56.443,-177.785,6.293,148.484
C00697=1203.840,184.547,-56.419,-177.788,6.291,148.485
C00698=1203.845,184.298,-56.395,-177.790,6.289,148.485
C00699=1203.849,184.048,-56.373,-177.793,6.287,148.485
C00700=1203.854,183.800,-56.350,-177.796,6.285,148.486
C00701=1203.859,183.551,-56.327,-177.798,6.284,148.486
C00702=1203.863,183.302,-56.304,-177.801,6.282,148.486
C00703=1203.868,183.053,-56.281,-177.804,6.280,148.487
C00704=1203.873,182.804,-56.258,-177.806,6.278,148.487
C00705=1203.877,182.555,-56.236,-177.808,6.277,148.487
C00706=1203.882,182.306,-56.213,-177.811,6.275,148.488
C00707=1203.886,182.057,-56.190,-177.814,6.274,148.488
C00708=1203.891,181.808,-56.167,-177.816,6.272,148.489
C00709=1203.895,181.560,-56.144,-177.819,6.270,148.489
C00710=1203.900,181.310,-56.122,-177.822,6.268,148.489
C00711=1203.904,181.062,-56.099,-177.824,6.266,148.490
C00712=1203.910,180.813,-56.076,-177.827,6.266,148.490
C00713=1203.915,180.564,-56.053,-177.830,6.264,148.491
C00714=1203.919,180.315,-56.031,-177.832,6.262,148.491
C00715=1203.924,180.065,-56.008,-177.835,6.260,148.491
C00716=1203.928,179.817,-55.986,-177.838,6.259,148.492
C00717=1203.933,179.568,-55.962,-177.840,6.257,148.492
C00718=1203.937,179.319,-55.940,-177.843,6.255,148.492
C00719=1203.942,179.071,-55.917,-177.845,6.254,148.493
C00720=1203.947,178.821,-55.895,-177.848,6.252,148.493
C00721=1203.951,178.572,-55.872,-177.850,6.250,148.493
C00722=1203.956,178.323,-55.850,-177.853,6.249,148.494
C00723=1203.960,178.075,-55.827,-177.856,6.247,148.494
C00724=1203.965,177.825,-55.805,-177.858,6.245,148.495
C00725=1203.969,177.576,-55.782,-177.861,6.243,148.495
C00726=1203.975,177.328,-55.760,-177.864,6.242,148.496
C00727=1203.979,177.079,-55.737,-177.866,6.241,148.496
C00728=1203.984,176.829,-55.714,-177.869,6.239,148.496
C00729=1203.988,176.581,-55.692,-177.872,6.237,148.497
C00730=1203.993,176.331,-55.669,-177.874,6.235,148.497
C00731=1203.997,176.083,-55.646,-177.877,6.233,148.497
C00732=1204.002,175.834,-55.625,-177.879,6.232,148.498
C00733=1204.007,175.585,-55.601,-177.882,6.231,148.498
C00734=1204.012,175.336,-55.580,-177.884,6.229,148.498
C00735=1204.016,175.087,-55.558,-177.887,6.227,148.499
C00736=1204.021,174.838,-55.534,-177.890,6.226,148.499
C00737=1204.026,174.589,-55.513,-177.893,6.224,148.500
C00738=1204.031,174.340,-55.490,-177.895,6.223,148.500
C00739=1204.035,174.091,-55.467,-177.898,6.221,148.500
C00740=1204.039,173.842,-55.446,-177.900,6.219,148.501
C00741=1204.044,173.593,-55.422,-177.903,6.217,148.501
C00742=1204.049,173.345,-55.401,-177.906,6.216,148.502
C00743=1204.053,173.095,-55.378,-177.908,6.215,148.502
C00744=1204.059,172.846,-55.356,-177.910,6.213,148.502
C00745=1204.063,172.598,-55.333,-177.913,6.211,148.503
C00746=1204.067,172.348,-55.311,-177.916,6.209,148.503
C00747=1204.072,172.100,-55.290,-177.919,6.208,148.504
C00748=1204.077,171.851,-55.266,-177.921,6.207,148.504
C00749=1204.082,171.602,-55.245,-177.924,6.205,148.504
C00750=1204.086,171.353,-55.223,-177.926,6.203,148.505
C00751=1204.091,171.104,-55.200,-177.929,6.201,148.505
C00752=1204.096,170.854,-55.178,-177.932,6.199,148.505
C00753=1204.100,170.606,-55.156,-177.934,6.199,148.506
C00754=1204.104,170.357,-55.134,-177.937,6.197,148.506
C00755=1204.109,170.107,-55.111,-177.939,6.195,148.507
C00756=1204.114,169.859,-55.090,-177.942,6.193,148.507
C00757=1204.119,169.609,-55.067,-177.945,6.192,148.508
C00758=1204.123,169.361,-55.045,-177.947,6.191,148.508
C00759=1204.127,169.112,-55.023,-177.950,6.189,148.508
C00760=1204.133,168.863,-55.001,-177.953,6.187,148.509
C00761=1204.137,168.614,-54.979,-177.955,6.186,148.509
C00762=1204.142,168.365,-54.957,-177.958,6.184,148.510
C00763=1204.146,168.116,-54.935,-177.960,6.183,148.510
C00764=1204.151,167.867,-54.913,-177.963,6.181,148.510
C00765=1204.156,167.618,-54.891,-177.966,6.179,148.511
C00766=1204.161,167.369,-54.869,-177.968,6.177,148.511
C00767=1204.165,167.120,-54.847,-177.971,6.177,148.512
C00768=1204.170,166.872,-54.825,-177.973,6.175,148.512
C00769=1204.174,166.622,-54.802,-177.976,6.173,148.512
C00770=1204.179,166.374,-54.781,-177.979,6.171,148.513
C00771=1204.183,166.124,-54.759,-177.981,6.170,148.513
C00772=1204.188,165.876,-54.737,-177.984,6.169,148.514
C00773=1204.194,165.627,-54.715,-177.987,6.167,148.514
C00774=1204.198,165.377,-54.693,-177.989,6.165,148.514
C00775=1204.203,165.129,-54.671,-177.992,6.164,148.515
C00776=1204.207,164.879,-54.649,-177.994,6.163,148.515
C00777=1204.212,164.631,-54.627,-177.997,6.161,148.516
C00778=1204.217,164.381,-54.606,-177.999,6.159,148.516
C00779=1204.222,164.132,-54.584,-178.003,6.157,148.517
C00780=1204.226,163.883,-54.562,-178.005,6.157,148.517
C00781=1204.231,163.634,-54.541,-178.007,6.155,148.517
C00782=1204.236,163.385,-54.519,-178.010,6.153,148.518
C00783=1204.240,163.136,-54.497,-178.013,6.151,148.518
C00784=1204.245,162.887,-54.475,-178.015,6.150,148.518
C00785=1204.249,162.638,-54.453,-178.018,6.149,148.519
C00786=1204.254,162.389,-54.431,-178.021,6.147,148.519
C00787=1204.259,162.141,-54.410,-178.023,6.145,148.520
C00788=1204.263,161.891,-54.388,-178.025,6.144,148.520
C00789=1204.268,161.642,-54.367,-178.028,6.142,148.521
C00790=1204.273,161.393,-54.345,-178.031,6.141,148.521
C00791=1204.277,161.144,-54.323,-178.034,6.139,148.522
C00792=1204.282,160.896,-54.301,-178.036,6.138,148.522
C00793=1204.287,160.646,-54.280,-178.039,6.136,148.522
C00794=1204.292,160.397,-54.258,-178.041,6.135,148.523
C00795=1204.297,160.148,-54.237,-178.044,6.134,148.523
C00796=1204.301,159.899,-54.215,-178.047,6.132,148.524
C00797=1204.306,159.650,-54.194,-178.049,6.130,148.524
C00798=1204.310,159.381,-54.170,-178.052,6.128,148.524
C00799=1204.316,159.112,-54.147,-178.055,6.127,148.525
C00800=1204.321,158.843,-54.123,-178.058,6.125,148.525
C00801=1204.326,158.574,-54.100,-178.060,6.123,148.526
C00802=1204.331,158.325,-54.079,-178.063,6.123,148.526
C00803=1204.335,158.076,-54.057,-178.066,6.121,148.527
C00804=1204.340,157.827,-54.035,-178.068,6.119,148.527
C00805=1204.345,157.578,-54.014,-178.071,6.117,148.527
C00806=1204.350,157.328,-53.992,-178.074,6.117,148.528
C00807=1204.354,157.080,-53.971,-178.076,6.115,148.528
C00808=1204.359,156.831,-53.950,-178.079,6.113,148.529
C00809=1204.363,156.581,-53.928,-178.081,6.112,148.529
C00810=1204.368,156.333,-53.906,-178.084,6.110,148.530
C00811=1204.373,156.084,-53.885,-178.087,6.109,148.530
C00812=1204.378,155.835,-53.864,-178.089,6.108,148.531
C00813=1204.382,155.585,-53.843,-178.092,6.106,148.531
C00814=1204.387,155.337,-53.821,-178.094,6.104,148.531
C00815=1204.392,155.087,-53.800,-178.098,6.103,148.532
C00816=1204.397,154.839,-53.779,-178.100,6.102,148.532
C00817=1204.401,154.589,-53.757,-178.102,6.100,148.533
C00818=1204.406,154.340,-53.736,-178.105,6.098,148.533
C00819=1204.410,154.092,-53.715,-178.107,6.097,148.533
C00820=1204.416,153.843,-53.694,-178.110,6.096,148.534
C00821=1204.420,153.593,-53.672,-178.113,6.094,148.534
C00822=1204.425,153.344,-53.651,-178.115,6.093,148.535
C00823=1204.429,153.096,-53.630,-178.118,6.091,148.535
C00824=1204.434,152.846,-53.609,-178.121,6.090,148.536
C00825=1204.439,152.596,-53.587,-178.123,6.089,148.536
C00826=1204.444,152.348,-53.566,-178.126,6.087,148.537
C00827=1204.448,152.099,-53.545,-178.128,6.085,148.537
C00828=1204.453,151.850,-53.524,-178.131,6.085,148.538
C00829=1204.458,151.601,-53.503,-178.134,6.083,148.538
C00830=1204.462,151.352,-53.481,-178.136,6.081,148.538
C00831=1204.467,151.103,-53.460,-178.138,6.080,148.539
C00832=1204.472,150.853,-53.439,-178.142,6.079,148.539
C00833=1204.477,150.605,-53.417,-178.144,6.077,148.540
C00834=1204.481,150.356,-53.397,-178.146,6.076,148.540
C00835=1204.486,150.106,-53.376,-178.149,6.074,148.540
C00836=1204.491,149.857,-53.354,-178.152,6.073,148.541
C00837=1204.495,149.608,-53.334,-178.154,6.072,148.541
C00838=1204.501,149.359,-53.313,-178.157,6.070,148.542
C00839=1204.505,149.110,-53.291,-178.160,6.069,148.542
C00840=1204.510,148.861,-53.271,-178.162,6.068,148.543
C00841=1204.514,148.611,-53.249,-178.165,6.066,148.543
C00842=1204.519,148.363,-53.228,-178.168,6.064,148.544
C00843=1204.524,148.114,-53.207,-178.170,6.063,148.544
C00844=1204.529,147.865,-53.186,-178.173,6.062,148.545
C00845=1204.533,147.616,-53.166,-178.176,6.060,148.545
C00846=1204.538,147.367,-53.144,-178.178,6.059,148.545
C00847=1204.543,147.118,-53.124,-178.181,6.058,148.546
C00848=1204.547,146.868,-53.103,-178.184,6.056,148.546
C00849=1204.552,146.619,-53.082,-178.186,6.055,148.547
C00850=1204.556,146.370,-53.061,-178.189,6.053,148.547
C00851=1204.562,146.121,-53.040,-178.191,6.052,148.548
C00852=1204.566,145.872,-53.019,-178.194,6.051,148.548
C00853=1204.571,145.623,-52.998,-178.196,6.049,148.548
C00854=1204.576,145.374,-52.978,-178.199,6.048,148.549
C00855=1204.581,145.125,-52.957,-178.202,6.046,148.549
C00856=1204.585,144.876,-52.936,-178.204,6.045,148.550
C00857=1204.590,144.626,-52.914,-178.207,6.044,148.550
C00858=1204.594,144.378,-52.894,-178.210,6.042,148.551
C00859=1204.599,144.128,-52.873,-178.212,6.040,148.551
C00860=1204.604,143.879,-52.853,-178.214,6.039,148.552
C00861=1204.609,143.630,-52.832,-178.217,6.038,148.552
C00862=1204.613,143.381,-52.811,-178.220,6.037,148.553
C00863=1204.618,143.132,-52.790,-178.222,6.035,148.553
C00864=1204.623,142.883,-52.770,-178.225,6.034,148.554
C00865=1204.628,142.634,-52.749,-178.228,6.033,148.554
C00866=1204.632,142.385,-52.729,-178.230,6.031,148.554
C00867=1204.638,142.135,-52.708,-178.233,6.030,148.555
C00868=1204.642,141.886,-52.687,-178.235,6.029,148.555
C00869=1204.647,141.637,-52.666,-178.238,6.027,148.556
C00870=1204.652,141.388,-52.646,-178.241,6.026,148.556
C00871=1204.656,141.139,-52.626,-178.243,6.024,148.557
C00872=1204.661,140.890,-52.605,-178.246,6.024,148.557
C00873=1204.666,140.641,-52.584,-178.249,6.022,148.558
C00874=1204.671,140.392,-52.563,-178.251,6.020,148.558
C00875=1204.675,140.143,-52.543,-178.254,6.019,148.559
C00876=1204.680,139.894,-52.523,-178.256,6.018,148.559
C00877=1204.685,139.645,-52.502,-178.259,6.017,148.560
C00878=1204.689,139.396,-52.481,-178.261,6.015,148.560
C00879=1204.694,139.147,-52.461,-178.264,6.013,148.560
C00880=1204.699,138.898,-52.440,-178.267,6.013,148.561
C00881=1204.703,138.649,-52.420,-178.269,6.011,148.561
C00882=1204.709,138.399,-52.399,-178.272,6.010,148.562
C00883=1204.713,138.150,-52.378,-178.275,6.009,148.562
C00884=1204.718,137.901,-52.359,-178.277,6.007,148.563
C00885=1204.723,137.652,-52.338,-178.280,6.006,148.563
C00886=1204.727,137.403,-52.317,-178.283,6.004,148.564
C00887=1204.732,137.154,-52.297,-178.285,6.003,148.564
C00888=1204.736,136.905,-52.277,-178.288,6.002,148.565
C00889=1204.741,136.655,-52.256,-178.291,6.000,148.565
C00890=1204.746,136.406,-52.236,-178.293,5.999,148.566
C00891=1204.751,136.157,-52.216,-178.296,5.998,148.566
C00892=1204.756,135.908,-52.195,-178.298,5.997,148.567
C00893=1204.760,135.659,-52.174,-178.301,5.995,148.567
C00894=1204.765,135.409,-52.155,-178.303,5.994,148.568
C00895=1204.769,135.160,-52.134,-178.306,5.993,148.568
C00896=1204.775,134.911,-52.113,-178.308,5.992,148.568
C00897=1204.780,134.663,-52.093,-178.311,5.990,148.569
C00898=1204.784,134.413,-52.074,-178.314,5.989,148.569
C00899=1204.789,134.164,-52.053,-178.316,5.988,148.570
C00900=1204.794,133.915,-52.032,-178.319,5.986,148.570
C00901=1204.798,133.666,-52.012,-178.321,5.985,148.571
C00902=1204.803,133.397,-51.991,-178.325,5.984,148.571
C00903=1204.809,133.128,-51.969,-178.327,5.982,148.572
C00904=1204.814,132.860,-51.947,-178.330,5.981,148.572
C00905=1204.819,132.591,-51.926,-178.333,5.980,148.573
C00906=1204.824,132.342,-51.905,-178.336,5.978,148.573
C00907=1204.829,132.093,-51.884,-178.338,5.977,148.574
C00908=1204.834,131.844,-51.865,-178.341,5.975,148.574
C00909=1204.838,131.595,-51.844,-178.344,5.974,148.575
C00910=1204.843,131.345,-51.825,-178.346,5.973,148.575
C00911=1204.847,131.096,-51.804,-178.349,5.971,148.576
C00912=1204.852,130.848,-51.784,-178.351,5.971,148.576
C00913=1204.857,130.598,-51.765,-178.354,5.969,148.577
C00914=1204.862,130.349,-51.744,-178.356,5.968,148.577
C00915=1204.867,130.099,-51.724,-178.359,5.966,148.578
C00916=1204.871,129.851,-51.704,-178.361,5.966,148.578
C00917=1204.876,129.601,-51.684,-178.364,5.964,148.579
C00918=1204.881,129.353,-51.664,-178.366,5.963,148.579
C00919=1204.886,129.103,-51.644,-178.370,5.962,148.580
C00920=1204.890,128.854,-51.624,-178.372,5.961,148.580
C00921=1204.895,128.605,-51.604,-178.374,5.959,148.581
C00922=1204.900,128.356,-51.584,-178.377,5.958,148.581
C00923=1204.905,128.107,-51.564,-178.380,5.957,148.582
C00924=1204.909,127.858,-51.544,-178.382,5.956,148.582
C00925=1204.915,127.608,-51.524,-178.385,5.954,148.583
C00926=1204.919,127.359,-51.504,-178.388,5.952,148.583
C00927=1204.924,127.109,-51.484,-178.390,5.952,148.584
C00928=1204.929,126.861,-51.465,-178.393,5.950,148.584
C00929=1204.934,126.612,-51.444,-178.395,5.949,148.584
C00930=1204.938,126.362,-51.425,-178.398,5.948,148.585
C00931=1204.943,126.113,-51.404,-178.400,5.947,148.585
C00932=1204.948,125.864,-51.385,-178.404,5.945,148.586
C00933=1204.953,125.615,-51.365,-178.406,5.944,148.586
C00934=1204.957,125.366,-51.345,-178.408,5.943,148.587
C00935=1204.962,125.116,-51.325,-178.411,5.942,148.588
C00936=1204.967,124.867,-51.305,-178.414,5.940,148.588
C00937=1204.972,124.618,-51.286,-178.416,5.940,148.589
C00938=1204.977,124.369,-51.266,-178.419,5.938,148.589
C00939=1204.981,124.119,-51.246,-178.422,5.937,148.590
C00940=1204.986,123.871,-51.227,-178.424,5.935,148.590
C00941=1204.991,123.622,-51.207,-178.426,5.935,148.590
C00942=1204.995,123.372,-51.187,-178.430,5.933,148.591
C00943=1205.000,123.123,-51.167,-178.432,5.932,148.591
C00944=1205.005,122.874,-51.148,-178.435,5.931,148.592
C00945=1205.010,122.625,-51.128,-178.437,5.930,148.592
C00946=1205.015,122.375,-51.109,-178.440,5.928,148.593
C00947=1205.020,122.127,-51.089,-178.442,5.927,148.593
C00948=1205.024,121.877,-51.069,-178.445,5.926,148.594
C00949=1205.029,121.628,-51.049,-178.448,5.925,148.594
C00950=1205.034,121.379,-51.030,-178.450,5.924,148.595
C00951=1205.038,121.130,-51.011,-178.453,5.923,148.596
C00952=1205.043,120.881,-50.990,-178.455,5.922,148.596
C00953=1205.048,120.632,-50.971,-178.458,5.920,148.597
C00954=1205.053,120.382,-50.952,-178.460,5.919,148.597
C00955=1205.058,120.133,-50.932,-178.463,5.918,148.597
C00956=1205.063,119.884,-50.913,-178.466,5.917,148.598
C00957=1205.068,119.634,-50.893,-178.468,5.915,148.598
C00958=1205.071,119.386,-50.873,-178.471,5.915,148.599
C00959=1205.077,119.137,-50.854,-178.474,5.913,148.599
C00960=1205.082,118.887,-50.834,-178.476,5.912,148.600
C00961=1205.086,118.638,-50.815,-178.479,5.910,148.600
C00962=1205.092,118.389,-50.795,-178.481,5.910,148.601
C00963=1205.096,118.139,-50.776,-178.484,5.908,148.601
C00964=1205.100,117.890,-50.757,-178.486,5.907,148.602
C00965=1205.106,117.641,-50.737,-178.490,5.906,148.603
C00966=1205.110,117.392,-50.718,-178.492,5.905,148.603
C00967=1205.116,117.143,-50.698,-178.494,5.904,148.604
C00968=1205.120,116.893,-50.679,-178.497,5.902,148.604
C00969=1205.125,116.644,-50.660,-178.500,5.902,148.605
C00970=1205.130,116.395,-50.640,-178.502,5.900,148.605
C00971=1205.135,116.145,-50.621,-178.505,5.899,148.606
C00972=1205.139,115.897,-50.602,-178.508,5.898,148.606
C00973=1205.144,115.647,-50.582,-178.510,5.897,148.606
C00974=1205.149,115.398,-50.563,-178.513,5.895,148.607
C00975=1205.154,115.149,-50.543,-178.515,5.894,148.607
C00976=1205.158,114.900,-50.524,-178.518,5.894,148.608
C00977=1205.163,114.651,-50.505,-178.520,5.892,148.609
C00978=1205.168,114.401,-50.485,-178.523,5.891,148.609
C00979=1205.173,114.153,-50.467,-178.526,5.890,148.610
C00980=1205.178,113.903,-50.447,-178.528,5.889,148.610
C00981=1205.183,113.654,-50.428,-178.531,5.887,148.611
C00982=1205.188,113.405,-50.408,-178.534,5.887,148.611
C00983=1205.192,113.155,-50.389,-178.536,5.886,148.612
C00984=1205.197,112.906,-50.370,-178.539,5.884,148.612
C00985=1205.202,112.656,-50.351,-178.541,5.883,148.613
C00986=1205.207,112.408,-50.332,-178.544,5.882,148.613
C00987=1205.211,112.158,-50.312,-178.546,5.881,148.614
C00988=1205.216,111.910,-50.294,-178.549,5.880,148.614
C00989=1205.221,111.660,-50.274,-178.552,5.879,148.615
C00990=1205.226,111.411,-50.255,-178.554,5.878,148.615
C00991=1205.230,111.161,-50.236,-178.557,5.876,148.616
C00992=1205.236,110.912,-50.217,-178.560,5.876,148.616
C00993=1205.240,110.663,-50.197,-178.562,5.874,148.617
C00994=1205.245,110.414,-50.179,-178.564,5.873,148.617
C00995=1205.250,110.165,-50.159,-178.568,5.872,148.618
C00996=1205.255,109.916,-50.141,-178.570,5.871,148.618
C00997=1205.259,109.666,-50.121,-178.572,5.870,148.619
C00998=1205.264,109.417,-50.103,-178.575,5.868,148.619
C00999=1205.269,109.168,-50.083,-178.578,5.868,148.620
C01000=1205.274,108.918,-50.065,-178.580,5.866,148.620
C01001=1205.278,108.669,-50.045,-178.583,5.865,148.621
C01002=1205.284,108.420,-50.026,-178.585,5.864,148.621
C01003=1205.288,108.170,-50.008,-178.588,5.863,148.622
C01004=1205.293,107.921,-49.989,-178.590,5.862,148.623
C01005=1205.298,107.673,-49.970,-178.593,5.861,148.623
C01006=1205.303,107.404,-49.949,-178.596,5.860,148.624
C01007=1205.309,107.136,-49.929,-178.599,5.858,148.624
C01008=1205.313,106.867,-49.909,-178.601,5.858,148.625
C01009=1205.319,106.599,-49.888,-178.605,5.856,148.625
C01010=1205.324,106.349,-49.869,-178.607,5.855,148.626
C01011=1205.328,106.100,-49.851,-178.610,5.854,148.627
C01012=1205.334,105.851,-49.831,-178.612,5.853,148.627
C01013=1205.338,105.601,-49.813,-178.615,5.852,148.628
C01014=1205.343,105.353,-49.794,-178.617,5.851,148.628
C01015=1205.347,105.103,-49.775,-178.620,5.850,148.629
C01016=1205.352,104.854,-49.757,-178.623,5.848,148.629
C01017=1205.358,104.605,-49.737,-178.625,5.848,148.630
C01018=1205.362,104.355,-49.719,-178.627,5.847,148.630
C01019=1205.367,104.106,-49.700,-178.631,5.845,148.631
C01020=1205.372,103.857,-49.681,-178.633,5.844,148.631
C01021=1205.376,103.608,-49.663,-178.635,5.844,148.632
C01022=1205.382,103.359,-49.644,-178.639,5.842,148.632
C01023=1205.386,103.109,-49.625,-178.641,5.842,148.633
C01024=1205.392,102.860,-49.606,-178.644,5.840,148.633
C01025=1205.396,102.611,-49.588,-178.646,5.839,148.634
C01026=1205.400,102.361,-49.569,-178.649,5.839,148.635
C01027=1205.406,102.112,-49.550,-178.651,5.837,148.635
C01028=1205.410,101.863,-49.532,-178.654,5.836,148.636
C01029=1205.415,101.614,-49.513,-178.656,5.835,148.636
C01030=1205.420,101.365,-49.495,-178.659,5.834,148.637
C01031=1205.425,101.115,-49.476,-178.661,5.833,148.637
C01032=1205.430,100.866,-49.457,-178.664,5.832,148.638
C01033=1205.435,100.617,-49.439,-178.667,5.831,148.638
C01034=1205.439,100.367,-49.420,-178.669,5.830,148.639
C01035=1205.445,100.118,-49.401,-178.672,5.828,148.639
C01036=1205.450,99.869,-49.383,-178.675,5.828,148.640
C01037=1205.454,99.619,-49.364,-178.677,5.827,148.640
C01038=1205.459,99.370,-49.346,-178.680,5.825,148.641
C01039=1205.464,99.121,-49.327,-178.683,5.825,148.642
C01040=1205.469,98.872,-49.309,-178.685,5.824,148.642
C01041=1205.473,98.622,-49.291,-178.688,5.822,148.643
C01042=1205.478,98.373,-49.271,-178.690,5.822,148.643
C01043=1205.483,98.124,-49.253,-178.693,5.821,148.644
C01044=1205.488,97.874,-49.235,-178.695,5.819,148.644
C01045=1205.493,97.626,-49.216,-178.698,5.819,148.645
C01046=1205.498,97.376,-49.198,-178.701,5.818,148.645
C01047=1205.503,97.127,-49.180,-178.703,5.816,148.646
C01048=1205.507,96.877,-49.161,-178.706,5.816,148.646
C01049=1205.512,96.628,-49.142,-178.708,5.815,148.647
C01050=1205.517,96.379,-49.124,-178.711,5.813,148.647
C01051=1205.522,96.129,-49.106,-178.713,5.812,148.648
C01052=1205.527,95.880,-49.088,-178.716,5.812,148.649
C01053=1205.531,95.632,-49.069,-178.719,5.810,148.649
C01054=1205.537,95.382,-49.051,-178.721,5.810,148.650
C01055=1205.542,95.133,-49.033,-178.724,5.809,148.650
C01056=1205.546,94.883,-49.014,-178.727,5.807,148.651
C01057=1205.551,94.634,-48.996,-178.729,5.807,148.651
C01058=1205.556,94.385,-48.978,-178.731,5.806,148.652
C01059=1205.561,94.136,-48.959,-178.735,5.804,148.652
C01060=1205.566,93.886,-48.941,-178.737,5.803,148.653
C01061=1205.570,93.637,-48.923,-178.739,5.803,148.653
C01062=1205.575,93.388,-48.905,-178.742,5.802,148.654
C01063=1205.580,93.139,-48.887,-178.745,5.800,148.654
C01064=1205.585,92.889,-48.869,-178.747,5.800,148.655
C01065=1205.589,92.639,-48.850,-178.749,5.799,148.656
C01066=1205.595,92.391,-48.831,-178.753,5.798,148.656
C01067=1205.600,92.141,-48.813,-178.755,5.797,148.657
C01068=1205.605,91.892,-48.795,-178.757,5.796,148.657
C01069=1205.610,91.643,-48.777,-178.761,5.795,148.658
C01070=1205.614,91.393,-48.759,-178.763,5.794,148.658
C01071=1205.619,91.144,-48.741,-178.765,5.793,148.659
C01072=1205.624,90.895,-48.723,-178.768,5.791,148.659
C01073=1205.629,90.646,-48.705,-178.771,5.791,148.660
C01074=1205.633,90.397,-48.687,-178.773,5.790,148.661
C01075=1205.638,90.147,-48.669,-178.775,5.789,148.661
C01076=1205.643,89.897,-48.651,-178.779,5.788,148.662
C01077=1205.648,89.648,-48.632,-178.781,5.787,148.662
C01078=1205.653,89.399,-48.614,-178.783,5.786,148.663
C01079=1205.658,89.150,-48.596,-178.786,5.785,148.663
C01080=1205.663,88.900,-48.578,-178.789,5.784,148.664
C01081=1205.668,88.651,-48.560,-178.791,5.784,148.665
C01082=1205.673,88.402,-48.542,-178.793,5.783,148.665
C01083=1205.677,88.152,-48.524,-178.797,5.781,148.666
C01084=1205.682,87.903,-48.506,-178.799,5.781,148.666
C01085=1205.687,87.654,-48.488,-178.801,5.780,148.667
C01086=1205.692,87.405,-48.470,-178.805,5.778,148.667
C01087=1205.697,87.156,-48.452,-178.807,5.777,148.668
C01088=1205.702,86.906,-48.435,-178.809,5.777,148.668
C01089=1205.707,86.657,-48.417,-178.812,5.776,148.669
C01090=1205.712,86.407,-48.399,-178.815,5.774,148.669
C01091=1205.717,86.158,-48.381,-178.817,5.774,148.670
C01092=1205.721,85.908,-48.362,-178.819,5.773,148.671
C01093=1205.726,85.659,-48.344,-178.822,5.772,148.671
C01094=1205.730,85.410,-48.327,-178.825,5.771,148.672
C01095=1205.735,85.161,-48.309,-178.827,5.770,148.672
C01096=1205.740,84.911,-48.292,-178.830,5.770,148.673
C01097=1205.745,84.662,-48.274,-178.833,5.768,148.673
C01098=1205.750,84.413,-48.256,-178.835,5.767,148.674
C01099=1205.755,84.164,-48.238,-178.838,5.767,148.675
C01100=1205.760,83.915,-48.220,-178.840,5.766,148.675
C01101=1205.765,83.665,-48.202,-178.843,5.764,148.676
C01102=1205.770,83.416,-48.184,-178.846,5.764,148.676
C01103=1205.775,83.166,-48.167,-178.848,5.763,148.677
C01104=1205.780,82.917,-48.149,-178.851,5.762,148.677
C01105=1205.784,82.668,-48.132,-178.853,5.761,148.678
C01106=1205.789,82.419,-48.114,-178.856,5.760,148.679
C01107=1205.794,82.169,-48.096,-178.859,5.759,148.679
C01108=1205.799,81.920,-48.078,-178.861,5.758,148.680
C01109=1205.804,81.670,-48.061,-178.864,5.757,148.680
C01110=1205.809,81.402,-48.041,-178.867,5.757,148.681
C01111=1205.815,81.133,-48.023,-178.869,5.756,148.682
C01112=1205.820,80.865,-48.003,-178.872,5.754,148.682
C01113=1205.825,80.597,-47.984,-178.874,5.754,148.683
C01114=1205.830,80.347,-47.967,-178.877,5.753,148.683
C01115=1205.834,80.098,-47.949,-178.880,5.752,148.684
C01116=1205.840,79.848,-47.932,-178.882,5.751,148.684
C01117=1205.845,79.599,-47.914,-178.885,5.750,148.685
C01118=1205.849,79.350,-47.896,-178.888,5.750,148.686
C01119=1205.854,79.101,-47.879,-178.890,5.748,148.686
C01120=1205.859,78.851,-47.861,-178.893,5.747,148.687
C01121=1205.864,78.602,-47.843,-178.895,5.746,148.687
C01122=1205.869,78.352,-47.826,-178.898,5.746,148.688
C01123=1205.874,78.103,-47.808,-178.901,5.744,148.689
C01124=1205.878,77.854,-47.791,-178.903,5.744,148.689
C01125=1205.883,77.605,-47.773,-178.906,5.743,148.690
C01126=1205.889,77.355,-47.756,-178.908,5.742,148.690
C01127=1205.894,77.106,-47.738,-178.911,5.741,148.691
C01128=1205.899,76.857,-47.722,-178.914,5.740,148.691
C01129=1205.903,76.608,-47.704,-178.916,5.740,148.692
C01130=1205.909,76.358,-47.687,-178.919,5.739,148.692
C01131=1205.913,76.109,-47.669,-178.921,5.738,148.693
C01132=1205.918,75.859,-47.652,-178.924,5.737,148.694
C01133=1205.923,75.610,-47.634,-178.926,5.736,148.694
C01134=1205.928,75.360,-47.617,-178.929,5.735,148.695
C01135=1205.932,75.111,-47.599,-178.932,5.735,148.695
C01136=1205.938,74.862,-47.582,-178.934,5.734,148.696
C01137=1205.942,74.612,-47.564,-178.937,5.732,148.697
C01138=1205.947,74.363,-47.547,-178.940,5.732,148.697
C01139=1205.952,74.114,-47.530,-178.942,5.731,148.698
C01140=1205.958,73.865,-47.512,-178.944,5.730,148.698
C01141=1205.962,73.616,-47.495,-178.947,5.730,148.699
C01142=1205.967,73.366,-47.478,-178.950,5.728,148.699
C01143=1205.972,73.116,-47.461,-178.952,5.727,148.700
C01144=1205.976,72.867,-47.443,-178.955,5.727,148.701
C01145=1205.982,72.617,-47.426,-178.957,5.726,148.701
C01146=1205.986,72.368,-47.409,-178.960,5.725,148.702
C01147=1205.992,72.120,-47.392,-178.963,5.724,148.702
C01148=1205.997,71.870,-47.374,-178.965,5.723,148.703
C01149=1206.001,71.621,-47.357,-178.968,5.723,148.704
C01150=1206.006,71.371,-47.340,-178.970,5.722,148.704
C01151=1206.011,71.122,-47.323,-178.973,5.721,148.705
C01152=1206.016,70.872,-47.305,-178.975,5.720,148.705
C01153=1206.021,70.623,-47.288,-178.978,5.719,148.706
C01154=1206.026,70.374,-47.272,-178.981,5.718,148.706
C01155=1206.031,70.124,-47.254,-178.983,5.718,148.707
C01156=1206.035,69.875,-47.237,-178.986,5.717,148.708
C01157=1206.041,69.625,-47.220,-178.988,5.716,148.708
C01158=1206.045,69.376,-47.203,-178.991,5.715,148.709
C01159=1206.050,69.126,-47.186,-178.994,5.714,148.709
C01160=1206.055,68.878,-47.169,-178.996,5.713,148.710
C01161=1206.060,68.628,-47.151,-178.999,5.713,148.711
C01162=1206.065,68.379,-47.135,-179.001,5.712,148.711
C01163=1206.070,68.129,-47.117,-179.003,5.711,148.712
C01164=1206.074,67.880,-47.100,-179.007,5.710,148.712
C01165=1206.080,67.631,-47.083,-179.009,5.709,148.713
C01166=1206.084,67.381,-47.066,-179.011,5.708,148.713
C01167=1206.090,67.132,-47.049,-179.014,5.708,148.714
C01168=1206.094,66.882,-47.033,-179.017,5.707,148.715
C01169=1206.099,66.633,-47.015,-179.019,5.707,148.715
C01170=1206.104,66.384,-46.998,-179.022,5.705,148.716
C01171=1206.109,66.134,-46.981,-179.025,5.704,148.716
C01172=1206.114,65.885,-46.964,-179.027,5.704,148.717
C01173=1206.119,65.635,-46.947,-179.029,5.703,148.718
C01174=1206.124,65.386,-46.931,-179.032,5.702,148.718
C01175=1206.129,65.137,-46.914,-179.035,5.702,148.719
C01176=1206.134,64.887,-46.897,-179.037,5.700,148.719
C01177=1206.138,64.638,-46.879,-179.040,5.700,148.720
C01178=1206.144,64.389,-46.863,-179.043,5.699,148.721
C01179=1206.148,64.140,-46.846,-179.045,5.698,148.721
C01180=1206.154,63.890,-46.829,-179.047,5.698,148.722
C01181=1206.158,63.640,-46.812,-179.050,5.697,148.722
C01182=1206.163,63.392,-46.796,-179.053,5.696,148.723
C01183=1206.168,63.142,-46.778,-179.055,5.695,148.723
C01184=1206.173,62.892,-46.762,-179.058,5.694,148.724
C01185=1206.179,62.643,-46.745,-179.061,5.694,148.725
C01186=1206.183,62.394,-46.728,-179.063,5.693,148.725
C01187=1206.188,62.144,-46.711,-179.065,5.692,148.726
C01188=1206.193,61.894,-46.694,-179.068,5.692,148.727
C01189=1206.198,61.646,-46.678,-179.071,5.691,148.727
C01190=1206.202,61.396,-46.661,-179.073,5.689,148.728
C01191=1206.208,61.146,-46.644,-179.076,5.689,148.728
C01192=1206.213,60.898,-46.628,-179.079,5.688,148.729
C01193=1206.217,60.648,-46.611,-179.081,5.687,148.729
C01194=1206.222,60.398,-46.594,-179.083,5.687,148.730
C01195=1206.227,60.150,-46.577,-179.086,5.686,148.731
C01196=1206.232,59.900,-46.561,-179.089,5.686,148.731
C01197=1206.237,59.650,-46.544,-179.091,5.685,148.732
C01198=1206.243,59.401,-46.528,-179.094,5.683,148.733
C01199=1206.247,59.151,-46.511,-179.097,5.683,148.733
C01200=1206.252,58.902,-46.494,-179.099,5.682,148.734
C01201=1206.257,58.653,-46.478,-179.101,5.681,148.734
C01202=1206.262,58.403,-46.461,-179.104,5.681,148.735
C01203=1206.266,58.154,-46.444,-179.107,5.680,148.736
C01204=1206.272,57.905,-46.427,-179.109,5.679,148.736
C01205=1206.277,57.655,-46.411,-179.111,5.679,148.737
C01206=1206.282,57.406,-46.395,-179.114,5.678,148.737
C01207=1206.286,57.156,-46.379,-179.117,5.677,148.738
C01208=1206.292,56.907,-46.361,-179.119,5.676,148.738
C01209=1206.297,56.658,-46.345,-179.122,5.675,148.739
C01210=1206.301,56.408,-46.328,-179.125,5.675,148.740
C01211=1206.306,56.158,-46.312,-179.127,5.674,148.740
C01212=1206.312,55.909,-46.295,-179.130,5.673,148.741
C01213=1206.316,55.660,-46.279,-179.132,5.673,148.742
C01214=1206.322,55.392,-46.261,-179.135,5.672,148.742
C01215=1206.326,55.123,-46.244,-179.138,5.671,148.743
C01216=1206.332,54.855,-46.226,-179.141,5.670,148.744
C01217=1206.338,54.586,-46.208,-179.143,5.670,148.744
C01218=1206.343,54.336,-46.192,-179.146,5.669,148.745
C01219=1206.348,54.088,-46.175,-179.148,5.668,148.745
C01220=1206.352,53.838,-46.159,-179.151,5.667,148.746
C01221=1206.357,53.588,-46.143,-179.154,5.667,148.747
C01222=1206.363,53.339,-46.126,-179.156,5.666,148.747
C01223=1206.367,53.089,-46.109,-179.159,5.665,148.748
C01224=1206.373,52.840,-46.094,-179.161,5.665,148.748
C01225=1206.377,52.591,-46.077,-179.164,5.664,148.749
C01226=1206.382,52.342,-46.061,-179.166,5.663,148.750
C01227=1206.387,52.092,-46.045,-179.169,5.663,148.750
C01228=1206.392,51.843,-46.028,-179.171,5.662,148.751
C01229=1206.397,51.593,-46.012,-179.174,5.661,148.752
C01230=1206.401,51.343,-45.996,-179.176,5.661,148.752
C01231=1206.407,51.094,-45.979,-179.179,5.659,148.753
C01232=1206.412,50.844,-45.963,-179.182,5.659,148.753
C01233=1206.417,50.595,-45.947,-179.185,5.658,148.754
C01234=1206.421,50.346,-45.930,-179.187,5.657,148.754
C01235=1206.427,50.096,-45.914,-179.189,5.657,148.755
C01236=1206.431,49.847,-45.898,-179.192,5.656,148.756
C01237=1206.437,49.598,-45.882,-179.195,5.656,148.756
C01238=1206.441,49.348,-45.865,-179.197,5.655,148.757
C01239=1206.447,49.099,-45.850,-179.199,5.654,148.758
C01240=1206.451,48.849,-45.833,-179.202,5.654,148.758
C01241=1206.456,48.600,-45.818,-179.205,5.653,148.759
C01242=1206.461,48.350,-45.801,-179.207,5.653,148.760
C01243=1206.466,48.101,-45.785,-179.210,5.652,148.760
C01244=1206.471,47.851,-45.769,-179.212,5.651,148.761
C01245=1206.476,47.602,-45.753,-179.215,5.651,148.761
C01246=1206.481,47.353,-45.736,-179.218,5.649,148.762
C01247=1206.486,47.103,-45.721,-179.220,5.648,148.762
C01248=1206.490,46.854,-45.704,-179.223,5.648,148.763
C01249=1206.496,46.604,-45.688,-179.225,5.647,148.764
C01250=1206.501,46.355,-45.672,-179.228,5.647,148.764
C01251=1206.506,46.105,-45.656,-179.230,5.646,148.765
C01252=1206.511,45.857,-45.640,-179.233,5.645,148.766
C01253=1206.516,45.606,-45.624,-179.236,5.645,148.766
C01254=1206.521,45.358,-45.608,-179.238,5.644,148.767
C01255=1206.525,45.108,-45.592,-179.240,5.643,148.767
C01256=1206.531,44.858,-45.576,-179.243,5.643,148.768
C01257=1206.535,44.609,-45.559,-179.246,5.642,148.769
C01258=1206.541,44.359,-45.544,-179.248,5.642,148.769
C01259=1206.546,44.111,-45.528,-179.251,5.641,148.770
C01260=1206.551,43.860,-45.512,-179.253,5.640,148.771
C01261=1206.556,43.611,-45.496,-179.256,5.640,148.771
C01262=1206.560,43.362,-45.480,-179.258,5.639,148.772
C01263=1206.565,43.112,-45.464,-179.261,5.639,148.773
C01264=1206.570,42.863,-45.449,-179.263,5.638,148.773
C01265=1206.575,42.614,-45.432,-179.266,5.637,148.774
C01266=1206.580,42.364,-45.417,-179.268,5.637,148.774
C01267=1206.585,42.114,-45.401,-179.272,5.635,148.775
C01268=1206.590,41.865,-45.384,-179.274,5.635,148.776
C01269=1206.596,41.616,-45.369,-179.276,5.634,148.776
C01270=1206.600,41.366,-45.353,-179.279,5.633,148.777
C01271=1206.605,41.117,-45.338,-179.282,5.633,148.777
C01272=1206.610,40.868,-45.321,-179.284,5.632,148.778
C01273=1206.615,40.618,-45.305,-179.286,5.631,148.779
C01274=1206.620,40.368,-45.290,-179.289,5.631,148.779
C01275=1206.626,40.119,-45.274,-179.292,5.630,148.780
C01276=1206.630,39.869,-45.258,-179.294,5.630,148.781
C01277=1206.635,39.620,-45.243,-179.297,5.629,148.781
C01278=1206.640,39.370,-45.227,-179.299,5.628,148.782
C01279=1206.645,39.121,-45.211,-179.302,5.628,148.782
C01280=1206.650,38.871,-45.196,-179.304,5.627,148.783
C01281=1206.655,38.622,-45.179,-179.307,5.627,148.784
C01282=1206.659,38.373,-45.164,-179.310,5.626,148.784
C01283=1206.665,38.124,-45.148,-179.312,5.625,148.785
C01284=1206.670,37.874,-45.133,-179.315,5.625,148.786
C01285=1206.675,37.624,-45.117,-179.317,5.624,148.786
C01286=1206.680,37.375,-45.101,-179.320,5.624,148.787
C01287=1206.685,37.126,-45.085,-179.322,5.623,148.788
C01288=1206.690,36.876,-45.069,-179.325,5.622,148.788
C01289=1206.695,36.627,-45.054,-179.327,5.622,148.789
C01290=1206.700,36.377,-45.038,-179.330,5.621,148.789
C01291=1206.704,36.127,-45.023,-179.333,5.621,148.790
C01292=1206.710,35.878,-45.007,-179.335,5.620,148.790
C01293=1206.715,35.629,-44.992,-179.337,5.619,148.791
C01294=1206.721,35.379,-44.976,-179.340,5.619,148.792
C01295=1206.725,35.129,-44.961,-179.343,5.618,148.793
C01296=1206.730,34.880,-44.945,-179.345,5.618,148.793
C01297=1206.735,34.631,-44.929,-179.347,5.617,148.794
C01298=1206.739,34.381,-44.914,-179.350,5.616,148.794
C01299=1206.744,34.132,-44.898,-179.353,5.616,148.795
C01300=1206.750,33.883,-44.882,-179.355,5.615,148.796
C01301=1206.755,33.634,-44.867,-179.358,5.615,148.796
C01302=1206.759,33.383,-44.851,-179.360,5.614,148.797
C01303=1206.765,33.134,-44.836,-179.363,5.613,148.797
C01304=1206.769,32.885,-44.821,-179.365,5.613,148.798
C01305=1206.775,32.636,-44.805,-179.368,5.612,148.799
C01306=1206.780,32.385,-44.789,-179.371,5.612,148.799
C01307=1206.784,32.136,-44.774,-179.373,5.611,148.800
C01308=1206.790,31.887,-44.759,-179.375,5.610,148.801
C01309=1206.795,31.638,-44.743,-179.378,5.610,148.801
C01310=1206.800,31.388,-44.729,-179.381,5.609,148.802
C01311=1206.805,31.138,-44.713,-179.383,5.609,148.803
C01312=1206.809,30.889,-44.698,-179.386,5.608,148.803
C01313=1206.815,30.639,-44.682,-179.388,5.607,148.804
C01314=1206.820,30.390,-44.667,-179.391,5.607,148.804
C01315=1206.824,30.140,-44.651,-179.394,5.606,148.805
C01316=1206.830,29.891,-44.636,-179.396,5.606,148.806
C01317=1206.834,29.642,-44.621,-179.399,5.605,148.806
C01318=1206.840,29.372,-44.604,-179.401,5.605,148.807
C01319=1206.846,29.104,-44.587,-179.404,5.604,148.808
C01320=1206.851,28.835,-44.572,-179.407,5.604,148.809
C01321=1206.856,28.567,-44.555,-179.409,5.603,148.809
C01322=1206.862,28.317,-44.539,-179.412,5.602,148.810
C01323=1206.866,28.068,-44.524,-179.414,5.602,148.810
C01324=1206.871,27.817,-44.509,-179.417,5.601,148.811
C01325=1206.876,27.568,-44.494,-179.419,5.601,148.812
C01326=1206.881,27.319,-44.478,-179.422,5.600,148.812
C01327=1206.886,27.070,-44.463,-179.425,5.600,148.813
C01328=1206.892,26.821,-44.448,-179.427,5.599,148.814
C01329=1206.896,26.571,-44.434,-179.430,5.598,148.814
C01330=1206.901,26.321,-44.418,-179.432,5.598,148.815
C01331=1206.906,26.072,-44.403,-179.435,5.597,148.816
C01332=1206.911,25.822,-44.387,-179.438,5.597,148.816
C01333=1206.916,25.573,-44.372,-179.440,5.596,148.817
C01334=1206.922,25.323,-44.357,-179.442,5.595,148.817
C01335=1206.926,25.074,-44.342,-179.445,5.595,148.818
C01336=1206.932,24.825,-44.327,-179.447,5.595,148.819
C01337=1206.936,24.574,-44.312,-179.450,5.594,148.819
C01338=1206.941,24.325,-44.296,-179.452,5.594,148.820
C01339=1206.946,24.076,-44.281,-179.455,5.593,148.821
C01340=1206.951,23.827,-44.266,-179.457,5.592,148.821
C01341=1206.956,23.577,-44.251,-179.460,5.592,148.822
C01342=1206.961,23.327,-44.236,-179.462,5.591,148.823
C01343=1206.966,23.078,-44.221,-179.465,5.591,148.823
C01344=1206.971,22.828,-44.207,-179.468,5.590,148.824
C01345=1206.977,22.579,-44.191,-179.470,5.590,148.825
C01346=1206.981,22.330,-44.176,-179.472,5.589,148.825
C01347=1206.986,22.079,-44.161,-179.475,5.588,148.826
C01348=1206.991,21.830,-44.146,-179.478,5.588,148.826
C01349=1206.996,21.580,-44.131,-179.480,5.587,148.827
C01350=1207.001,21.331,-44.116,-179.483,5.587,148.828
C01351=1207.006,21.082,-44.101,-179.486,5.586,148.828
C01352=1207.011,20.832,-44.087,-179.488,5.585,148.829
C01353=1207.016,20.583,-44.071,-179.490,5.586,148.830
C01354=1207.021,20.333,-44.057,-179.493,5.585,148.830
C01355=1207.026,20.084,-44.042,-179.495,5.585,148.831
C01356=1207.031,19.835,-44.026,-179.498,5.584,148.832
C01357=1207.036,19.585,-44.012,-179.501,5.584,148.832
C01358=1207.042,19.335,-43.996,-179.503,5.583,148.833
C01359=1207.047,19.086,-43.982,-179.505,5.582,148.833
C01360=1207.051,18.837,-43.967,-179.508,5.582,148.834
C01361=1207.057,18.587,-43.952,-179.511,5.581,148.835
C01362=1207.062,18.338,-43.937,-179.513,5.581,148.835
C01363=1207.067,18.088,-43.923,-179.516,5.580,148.836
C01364=1207.071,17.839,-43.908,-179.518,5.579,148.837
C01365=1207.077,17.589,-43.893,-179.521,5.579,148.837
C01366=1207.082,17.340,-43.878,-179.523,5.579,148.838
C01367=1207.087,17.090,-43.864,-179.525,5.579,148.839
C01368=1207.092,16.840,-43.848,-179.528,5.578,148.839
C01369=1207.097,16.591,-43.834,-179.531,5.578,148.840
C01370=1207.102,16.342,-43.819,-179.533,5.577,148.841
C01371=1207.107,16.092,-43.805,-179.536,5.576,148.841
C01372=1207.112,15.842,-43.790,-179.538,5.576,148.842
C01373=1207.117,15.593,-43.775,-179.541,5.575,148.843
C01374=1207.122,15.343,-43.760,-179.544,5.575,148.843
C01375=1207.127,15.094,-43.746,-179.546,5.574,148.844
C01376=1207.132,14.844,-43.731,-179.549,5.574,148.845
C01377=1207.137,14.594,-43.716,-179.550,5.574,148.845
C01378=1207.142,14.345,-43.701,-179.553,5.573,148.846
C01379=1207.147,14.096,-43.687,-179.556,5.573,148.846
C01380=1207.152,13.846,-43.671,-179.558,5.572,148.847
C01381=1207.157,13.596,-43.657,-179.561,5.572,148.848
C01382=1207.162,13.347,-43.643,-179.564,5.571,148.848
C01383=1207.167,13.098,-43.628,-179.566,5.570,148.849
C01384=1207.172,12.848,-43.614,-179.568,5.570,148.850
C01385=1207.177,12.598,-43.599,-179.571,5.569,148.850
C01386=1207.182,12.349,-43.584,-179.573,5.569,148.851
C01387=1207.187,12.099,-43.570,-179.576,5.569,148.852
C01388=1207.193,11.850,-43.556,-179.578,5.568,148.852
C01389=1207.197,11.601,-43.541,-179.581,5.568,148.853
C01390=1207.203,11.351,-43.526,-179.584,5.567,148.854
C01391=1207.208,11.101,-43.511,-179.586,5.566,148.854
C01392=1207.213,10.852,-43.497,-179.589,5.566,148.855
C01393=1207.217,10.602,-43.482,-179.591,5.565,148.856
C01394=1207.222,10.353,-43.468,-179.594,5.565,148.856
C01395=1207.227,10.103,-43.454,-179.596,5.565,148.857
C01396=1207.232,9.853,-43.439,-179.599,5.565,148.858
C01397=1207.237,9.604,-43.424,-179.601,5.564,148.858
C01398=1207.243,9.354,-43.410,-179.603,5.563,148.859
C01399=1207.248,9.105,-43.396,-179.606,5.563,148.859
C01400=1207.253,8.855,-43.381,-179.609,5.562,148.860
C01401=1207.258,8.606,-43.367,-179.611,5.562,148.861
C01402=1207.263,8.357,-43.352,-179.614,5.561,148.861
C01403=1207.268,8.107,-43.338,-179.616,5.562,148.862
C01404=1207.273,7.857,-43.323,-179.619,5.561,148.863
C01405=1207.278,7.608,-43.309,-179.621,5.560,148.863
C01406=1207.283,7.359,-43.295,-179.624,5.560,148.864
C01407=1207.288,7.109,-43.281,-179.626,5.559,148.865
C01408=1207.293,6.860,-43.266,-179.629,5.559,148.865
C01409=1207.298,6.610,-43.252,-179.632,5.558,148.866
C01410=1207.303,6.360,-43.237,-179.634,5.558,148.867
C01411=1207.308,6.110,-43.223,-179.636,5.558,148.867
C01412=1207.313,5.861,-43.208,-179.638,5.557,148.868
C01413=1207.319,5.612,-43.194,-179.641,5.557,148.869
C01414=1207.324,5.362,-43.180,-179.644,5.556,148.869
C01415=1207.329,5.112,-43.166,-179.646,5.556,148.870
C01416=1207.334,4.862,-43.152,-179.649,5.555,148.871
C01417=1207.339,4.613,-43.137,-179.652,5.555,148.871
C01418=1207.343,4.364,-43.122,-179.654,5.555,148.872
C01419=1207.349,4.115,-43.108,-179.656,5.554,148.872
C01420=1207.354,3.865,-43.094,-179.659,5.554,148.873
C01421=1207.359,3.615,-43.080,-179.661,5.553,148.874
C01422=1207.364,3.346,-43.065,-179.664,5.553,148.874
C01423=1207.369,3.077,-43.049,-179.667,5.552,148.875
C01424=1207.375,2.808,-43.035,-179.670,5.552,148.876
C01425=1207.381,2.539,-43.020,-179.672,5.551,148.877
C01426=1207.386,2.289,-43.005,-179.674,5.551,148.877
C01427=1207.391,2.039,-42.991,-179.677,5.550,148.878
C01428=1207.396,1.790,-42.977,-179.679,5.550,148.879
C01429=1207.401,1.541,-42.963,-179.682,5.550,148.879
C01430=1207.406,1.291,-42.949,-179.684,5.549,148.880
C01431=1207.411,1.041,-42.934,-179.687,5.549,148.881
C01432=1207.416,0.792,-42.920,-179.690,5.548,148.881
C01433=1207.421,0.543,-42.907,-179.692,5.548,148.882
C01434=1207.426,0.293,-42.892,-179.695,5.547,148.883
C01435=1207.431,0.043,-42.878,-179.697,5.547,148.883
C01436=1207.436,-0.206,-42.864,-179.699,5.547,148.884
C01437=1207.441,-0.455,-42.850,-179.702,5.546,148.885
C01438=1207.446,-0.705,-42.836,-179.705,5.546,148.885
C01439=1207.451,-0.955,-42.821,-179.707,5.545,148.886
C01440=1207.457,-1.205,-42.808,-179.710,5.545,148.887
C01441=1207.462,-1.454,-42.794,-179.712,5.545,148.887
C01442=1207.466,-1.703,-42.780,-179.714,5.544,148.888
C01443=1207.471,-1.953,-42.766,-179.717,5.544,148.888
C01444=1207.477,-2.202,-42.752,-179.720,5.543,148.889
C01445=1207.482,-2.452,-42.738,-179.722,5.543,148.890
C01446=1207.487,-2.702,-42.723,-179.725,5.542,148.891
C01447=1207.492,-2.952,-42.710,-179.727,5.543,148.891
C01448=1207.497,-3.201,-42.697,-179.730,5.542,148.892
C01449=1207.502,-3.450,-42.682,-179.732,5.542,148.893
C01450=1207.507,-3.700,-42.668,-179.734,5.541,148.893
C01451=1207.512,-3.949,-42.654,-179.737,5.540,148.894
C01452=1207.518,-4.199,-42.641,-179.739,5.540,148.894
C01453=1207.523,-4.449,-42.626,-179.742,5.540,148.895
C01454=1207.527,-4.698,-42.613,-179.744,5.539,148.896
C01455=1207.532,-4.947,-42.599,-179.747,5.539,148.897
C01456=1207.537,-5.197,-42.584,-179.750,5.538,148.897
C01457=1207.543,-5.447,-42.571,-179.752,5.538,148.898
C01458=1207.548,-5.696,-42.557,-179.754,5.538,148.898
C01459=1207.552,-5.946,-42.543,-179.757,5.537,148.899
C01460=1207.558,-6.196,-42.530,-179.759,5.537,148.900
C01461=1207.563,-6.445,-42.516,-179.762,5.536,148.900
C01462=1207.568,-6.695,-42.501,-179.765,5.536,148.901
C01463=1207.573,-6.944,-42.488,-179.767,5.536,148.902
C01464=1207.578,-7.194,-42.475,-179.769,5.536,148.903
C01465=1207.583,-7.444,-42.460,-179.772,5.535,148.903
C01466=1207.588,-7.692,-42.447,-179.775,5.535,148.904
C01467=1207.593,-7.943,-42.433,-179.777,5.534,148.904
C01468=1207.598,-8.192,-42.419,-179.779,5.534,148.905
C01469=1207.604,-8.441,-42.405,-179.782,5.534,148.906
C01470=1207.608,-8.691,-42.392,-179.784,5.533,148.906
C01471=1207.614,-8.940,-42.378,-179.787,5.533,148.907
C01472=1207.619,-9.190,-42.364,-179.789,5.532,148.908
C01473=1207.623,-9.440,-42.351,-179.792,5.533,148.909
C01474=1207.629,-9.689,-42.337,-179.794,5.532,148.909
C01475=1207.634,-9.940,-42.324,-179.796,5.531,148.910
C01476=1207.639,-10.188,-42.310,-179.799,5.531,148.910
C01477=1207.644,-10.438,-42.296,-179.802,5.530,148.911
C01478=1207.649,-10.688,-42.283,-179.804,5.531,148.912
C01479=1207.654,-10.937,-42.269,-179.806,5.530,148.912
C01480=1207.659,-11.187,-42.256,-179.809,5.530,148.913
C01481=1207.665,-11.436,-42.242,-179.812,5.529,148.914
C01482=1207.669,-11.686,-42.229,-179.814,5.529,148.915
C01483=1207.674,-11.936,-42.214,-179.816,5.529,148.915
C01484=1207.680,-12.185,-42.201,-179.819,5.528,148.916
C01485=1207.684,-12.435,-42.188,-179.821,5.528,148.916
C01486=1207.690,-12.684,-42.174,-179.824,5.527,148.917
C01487=1207.694,-12.934,-42.161,-179.826,5.527,148.918
C01488=1207.700,-13.183,-42.147,-179.829,5.527,148.918
C01489=1207.705,-13.433,-42.133,-179.831,5.526,148.919
C01490=1207.710,-13.682,-42.120,-179.834,5.526,148.920
C01491=1207.715,-13.932,-42.106,-179.837,5.525,148.921
C01492=1207.719,-14.182,-42.093,-179.839,5.526,148.921
C01493=1207.725,-14.431,-42.080,-179.841,5.525,148.922
C01494=1207.730,-14.681,-42.065,-179.844,5.524,148.922
C01495=1207.735,-14.931,-42.053,-179.846,5.524,148.923
C01496=1207.741,-15.181,-42.039,-179.848,5.524,148.924
C01497=1207.745,-15.430,-42.026,-179.851,5.524,148.924
C01498=1207.751,-15.680,-42.012,-179.854,5.523,148.925
C01499=1207.756,-15.929,-41.999,-179.856,5.523,148.926
C01500=1207.761,-16.179,-41.985,-179.859,5.522,148.927
C01501=1207.766,-16.428,-41.973,-179.861,5.523,148.927
C01502=1207.771,-16.678,-41.958,-179.863,5.522,148.928
C01503=1207.777,-16.928,-41.945,-179.866,5.521,148.928
C01504=1207.781,-17.177,-41.932,-179.868,5.521,148.929
C01505=1207.787,-17.427,-41.918,-179.871,5.521,148.930
C01506=1207.791,-17.677,-41.905,-179.873,5.521,148.930
C01507=1207.797,-17.926,-41.891,-179.876,5.520,148.931
C01508=1207.801,-18.176,-41.879,-179.879,5.520,148.932
C01509=1207.807,-18.425,-41.865,-179.881,5.520,148.933
C01510=1207.812,-18.675,-41.852,-179.883,5.519,148.933
C01511=1207.817,-18.924,-41.838,-179.885,5.519,148.934
C01512=1207.822,-19.174,-41.825,-179.888,5.518,148.934
C01513=1207.827,-19.423,-41.812,-179.891,5.518,148.935
C01514=1207.833,-19.673,-41.799,-179.893,5.518,148.936
C01515=1207.837,-19.923,-41.786,-179.895,5.517,148.937
C01516=1207.843,-20.172,-41.772,-179.898,5.517,148.937
C01517=1207.847,-20.422,-41.759,-179.901,5.517,148.938
C01518=1207.853,-20.671,-41.746,-179.903,5.517,148.939
C01519=1207.858,-20.921,-41.733,-179.906,5.516,148.939
C01520=1207.863,-21.170,-41.719,-179.908,5.515,148.940
C01521=1207.868,-21.420,-41.706,-179.910,5.515,148.940
C01522=1207.874,-21.670,-41.693,-179.912,5.515,148.941
C01523=1207.879,-21.919,-41.680,-179.915,5.515,148.942
C01524=1207.883,-22.169,-41.667,-179.918,5.514,148.943
C01525=1207.889,-22.418,-41.653,-179.920,5.514,148.943
C01526=1207.894,-22.688,-41.640,-179.923,5.514,148.944
C01527=1207.899,-22.957,-41.625,-179.925,5.514,148.945
C01528=1207.905,-23.227,-41.611,-179.928,5.513,148.945
C01529=1207.910,-23.497,-41.597,-179.930,5.513,148.946
C01530=1207.916,-23.746,-41.584,-179.933,5.512,148.947
C01531=1207.921,-23.996,-41.570,-179.936,5.512,148.947
C01532=1207.926,-24.245,-41.558,-179.938,5.512,148.948
C01533=1207.931,-24.495,-41.544,-179.941,5.512,148.949
C01534=1207.936,-24.745,-41.531,-179.943,5.511,148.949
C01535=1207.941,-24.994,-41.519,-179.945,5.512,148.950
C01536=1207.946,-25.244,-41.505,-179.948,5.511,148.951
C01537=1207.951,-25.493,-41.492,-179.951,5.511,148.952
C01538=1207.956,-25.743,-41.479,-179.953,5.510,148.952
C01539=1207.962,-25.993,-41.466,-179.955,5.510,148.953
C01540=1207.967,-26.242,-41.453,-179.958,5.510,148.953
C01541=1207.971,-26.492,-41.440,-179.960,5.509,148.954
C01542=1207.977,-26.741,-41.427,-179.963,5.509,148.955
C01543=1207.982,-26.991,-41.414,-179.965,5.509,148.956
C01544=1207.987,-27.241,-41.402,-179.968,5.508,148.956
C01545=1207.993,-27.490,-41.388,-179.970,5.508,148.957
C01546=1207.998,-27.740,-41.376,-179.973,5.507,148.958
C01547=1208.002,-27.990,-41.363,-179.974,5.507,148.958
C01548=1208.007,-28.239,-41.350,-179.977,5.507,148.959
C01549=1208.013,-28.489,-41.337,-179.980,5.506,148.959
C01550=1208.018,-28.739,-41.324,-179.982,5.507,148.960
C01551=1208.023,-28.987,-41.311,-179.985,5.506,148.961
C01552=1208.028,-29.237,-41.298,-179.987,5.506,148.962
C01553=1208.033,-29.487,-41.285,-179.990,5.505,148.962
C01554=1208.038,-29.736,-41.272,-179.992,5.506,148.963
C01555=1208.043,-29.986,-41.259,-179.995,5.505,148.964
C01556=1208.048,-30.236,-41.246,-179.997,5.504,148.964
C01557=1208.054,-30.486,-41.234,-179.999,5.505,148.965
C01558=1208.059,-30.735,-41.221,179.998,5.504,148.966
C01559=1208.064,-30.985,-41.208,179.996,5.504,148.966
C01560=1208.069,-31.235,-41.196,179.993,5.503,148.967
C01561=1208.075,-31.484,-41.183,179.991,5.504,148.968
C01562=1208.080,-31.734,-41.170,179.988,5.503,148.968
C01563=1208.084,-31.984,-41.157,179.986,5.503,148.969
C01564=1208.089,-32.233,-41.144,179.984,5.503,148.970
C01565=1208.095,-32.482,-41.132,179.981,5.503,148.970
C01566=1208.099,-32.732,-41.119,179.979,5.502,148.971
C01567=1208.105,-32.982,-41.106,179.976,5.501,148.972
C01568=1208.110,-33.231,-41.093,179.974,5.502,148.972
C01569=1208.115,-33.481,-41.080,179.971,5.501,148.973
C01570=1208.120,-33.731,-41.068,179.969,5.501,148.974
C01571=1208.125,-33.980,-41.056,179.967,5.501,148.974
C01572=1208.130,-34.230,-41.043,179.964,5.500,148.975
C01573=1208.136,-34.479,-41.030,179.961,5.500,148.976
C01574=1208.141,-34.729,-41.017,179.959,5.500,148.976
C01575=1208.146,-34.979,-41.004,179.957,5.499,148.977
C01576=1208.151,-35.228,-40.992,179.954,5.499,148.978
C01577=1208.156,-35.478,-40.980,179.952,5.499,148.978
C01578=1208.161,-35.727,-40.967,179.950,5.499,148.979
C01579=1208.166,-35.977,-40.954,179.947,5.498,148.980
C01580=1208.172,-36.227,-40.941,179.944,5.498,148.980
C01581=1208.177,-36.476,-40.928,179.942,5.498,148.981
C01582=1208.182,-36.726,-40.916,179.940,5.498,148.982
C01583=1208.187,-36.976,-40.903,179.937,5.497,148.983
C01584=1208.192,-37.226,-40.891,179.935,5.498,148.983
C01585=1208.197,-37.475,-40.878,179.933,5.497,148.984
C01586=1208.203,-37.725,-40.866,179.930,5.496,148.984
C01587=1208.208,-37.974,-40.854,179.927,5.496,148.985
C01588=1208.212,-38.224,-40.841,179.925,5.496,148.986
C01589=1208.217,-38.473,-40.828,179.923,5.496,148.987
C01590=1208.223,-38.723,-40.816,179.920,5.495,148.987
C01591=1208.228,-38.973,-40.804,179.918,5.496,148.988
C01592=1208.234,-39.222,-40.791,179.915,5.495,148.989
C01593=1208.239,-39.472,-40.778,179.913,5.495,148.989
C01594=1208.244,-39.722,-40.766,179.911,5.495,148.990
C01595=1208.249,-39.972,-40.753,179.908,5.494,148.990
C01596=1208.254,-40.221,-40.740,179.906,5.494,148.991
C01597=1208.259,-40.471,-40.729,179.904,5.494,148.992
C01598=1208.264,-40.720,-40.716,179.901,5.494,148.993
C01599=1208.270,-40.970,-40.703,179.898,5.493,148.993
C01600=1208.274,-41.220,-40.691,179.896,5.493,148.994
C01601=1208.280,-41.469,-40.679,179.894,5.493,148.995
C01602=1208.285,-41.719,-40.666,179.891,5.493,148.995
C01603=1208.290,-41.969,-40.654,179.889,5.492,148.996
C01604=1208.295,-42.218,-40.641,179.887,5.492,148.997
C01605=1208.301,-42.468,-40.630,179.884,5.492,148.997
C01606=1208.306,-42.717,-40.617,179.882,5.492,148.998
C01607=1208.310,-42.967,-40.604,179.879,5.491,148.999
C01608=1208.315,-43.217,-40.593,179.877,5.491,148.999
C01609=1208.320,-43.466,-40.580,179.874,5.491,149.000
C01610=1208.326,-43.716,-40.568,179.872,5.491,149.001
C01611=1208.331,-43.966,-40.556,179.869,5.490,149.001
C01612=1208.336,-44.215,-40.543,179.868,5.490,149.002
C01613=1208.341,-44.465,-40.531,179.865,5.490,149.003
C01614=1208.346,-44.714,-40.519,179.862,5.489,149.003
C01615=1208.352,-44.964,-40.507,179.860,5.490,149.004
C01616=1208.357,-45.213,-40.494,179.857,5.489,149.005
C01617=1208.362,-45.464,-40.482,179.855,5.489,149.005
C01618=1208.367,-45.713,-40.469,179.853,5.489,149.006
C01619=1208.372,-45.963,-40.457,179.850,5.489,149.007
C01620=1208.377,-46.213,-40.445,179.847,5.488,149.008
C01621=1208.383,-46.463,-40.433,179.846,5.488,149.008
C01622=1208.387,-46.712,-40.421,179.843,5.488,149.009
C01623=1208.393,-46.961,-40.409,179.840,5.487,149.009
C01624=1208.398,-47.211,-40.396,179.838,5.488,149.010
C01625=1208.403,-47.461,-40.384,179.836,5.487,149.011
C01626=1208.408,-47.710,-40.372,179.833,5.487,149.012
C01627=1208.414,-47.960,-40.360,179.831,5.487,149.012
C01628=1208.419,-48.209,-40.347,179.828,5.487,149.013
C01629=1208.424,-48.459,-40.336,179.826,5.486,149.014
C01630=1208.430,-48.730,-40.323,179.824,5.486,149.014
C01631=1208.435,-48.999,-40.309,179.821,5.486,149.015
C01632=1208.441,-49.269,-40.296,179.818,5.486,149.016
C01633=1208.446,-49.539,-40.283,179.816,5.485,149.016
C01634=1208.451,-49.789,-40.271,179.813,5.485,149.017
C01635=1208.456,-50.039,-40.259,179.811,5.485,149.018
C01636=1208.462,-50.288,-40.247,179.808,5.485,149.019
C01637=1208.466,-50.537,-40.235,179.806,5.485,149.019
C01638=1208.472,-50.787,-40.223,179.804,5.484,149.020
C01639=1208.477,-51.037,-40.211,179.801,5.484,149.020
C01640=1208.482,-51.287,-40.199,179.799,5.484,149.021
C01641=1208.488,-51.537,-40.187,179.796,5.483,149.022
C01642=1208.492,-51.786,-40.175,179.794,5.483,149.023
C01643=1208.497,-52.036,-40.163,179.792,5.483,149.023
C01644=1208.503,-52.285,-40.151,179.789,5.483,149.024
C01645=1208.508,-52.535,-40.139,179.786,5.482,149.025
C01646=1208.513,-52.784,-40.127,179.784,5.483,149.025
C01647=1208.518,-53.034,-40.115,179.782,5.482,149.026
C01648=1208.524,-53.284,-40.103,179.780,5.482,149.027
C01649=1208.529,-53.534,-40.091,179.777,5.482,149.027
C01650=1208.533,-53.783,-40.079,179.775,5.481,149.028
C01651=1208.539,-54.033,-40.067,179.773,5.482,149.029
C01652=1208.544,-54.283,-40.056,179.770,5.481,149.029
C01653=1208.549,-54.532,-40.044,179.767,5.481,149.030
C01654=1208.554,-54.782,-40.032,179.765,5.481,149.031
C01655=1208.559,-55.032,-40.020,179.763,5.480,149.031
C01656=1208.565,-55.282,-40.008,179.761,5.481,149.032
C01657=1208.569,-55.531,-39.996,179.758,5.480,149.033
C01658=1208.575,-55.781,-39.984,179.756,5.480,149.033
C01659=1208.580,-56.031,-39.972,179.754,5.480,149.034
C01660=1208.585,-56.280,-39.961,179.751,5.480,149.035
C01661=1208.590,-56.530,-39.949,179.748,5.479,149.035
C01662=1208.595,-56.780,-39.936,179.746,5.480,149.036
C01663=1208.601,-57.029,-39.925,179.744,5.479,149.037
C01664=1208.606,-57.279,-39.914,179.741,5.478,149.037
C01665=1208.612,-57.529,-39.902,179.739,5.479,149.038
C01666=1208.616,-57.778,-39.890,179.736,5.478,149.039
C01667=1208.621,-58.027,-39.878,179.734,5.479,149.039
C01668=1208.627,-58.277,-39.866,179.732,5.478,149.040
C01669=1208.631,-58.527,-39.855,179.729,5.478,149.041
C01670=1208.637,-58.777,-39.843,179.727,5.478,149.042
C01671=1208.642,-59.027,-39.831,179.724,5.478,149.042
C01672=1208.647,-59.277,-39.819,179.723,5.477,149.043
C01673=1208.652,-59.526,-39.808,179.720,5.477,149.043
C01674=1208.657,-59.775,-39.796,179.717,5.477,149.044
C01675=1208.663,-60.025,-39.784,179.715,5.477,149.045
C01676=1208.668,-60.275,-39.772,179.713,5.476,149.046
C01677=1208.673,-60.524,-39.761,179.710,5.476,149.046
C01678=1208.678,-60.774,-39.749,179.708,5.476,149.047
C01679=1208.683,-61.024,-39.738,179.706,5.476,149.047
C01680=1208.689,-61.274,-39.726,179.704,5.476,149.048
C01681=1208.693,-61.523,-39.715,179.701,5.475,149.049
C01682=1208.699,-61.773,-39.703,179.698,5.475,149.050
C01683=1208.705,-62.023,-39.691,179.696,5.475,149.050
C01684=1208.709,-62.272,-39.680,179.694,5.475,149.051
C01685=1208.715,-62.522,-39.668,179.691,5.475,149.052
C01686=1208.720,-62.772,-39.657,179.689,5.475,149.052
C01687=1208.725,-63.022,-39.645,179.687,5.474,149.053
C01688=1208.730,-63.271,-39.634,179.685,5.474,149.054
C01689=1208.735,-63.521,-39.622,179.682,5.474,149.054
C01690=1208.740,-63.770,-39.611,179.680,5.474,149.055
C01691=1208.746,-64.020,-39.599,179.677,5.474,149.056
C01692=1208.750,-64.270,-39.588,179.674,5.473,149.056
C01693=1208.756,-64.520,-39.576,179.672,5.474,149.057
C01694=1208.761,-64.769,-39.564,179.670,5.473,149.058
C01695=1208.766,-65.019,-39.552,179.668,5.473,149.058
C01696=1208.771,-65.268,-39.542,179.665,5.473,149.059
C01697=1208.777,-65.518,-39.530,179.663,5.472,149.060
C01698=1208.781,-65.768,-39.518,179.661,5.473,149.060
C01699=1208.787,-66.018,-39.506,179.658,5.472,149.061
C01700=1208.792,-66.267,-39.495,179.656,5.473,149.062
C01701=1208.798,-66.516,-39.484,179.653,5.472,149.063
C01702=1208.802,-66.766,-39.472,179.651,5.471,149.063
C01703=1208.808,-67.016,-39.460,179.649,5.472,149.064
C01704=1208.812,-67.266,-39.449,179.646,5.471,149.064
C01705=1208.818,-67.516,-39.438,179.644,5.472,149.065
C01706=1208.823,-67.765,-39.427,179.642,5.471,149.066
C01707=1208.829,-68.015,-39.415,179.639,5.471,149.067
C01708=1208.834,-68.265,-39.404,179.637,5.471,149.067
C01709=1208.839,-68.515,-39.392,179.635,5.470,149.068
C01710=1208.844,-68.764,-39.381,179.633,5.471,149.068
C01711=1208.849,-69.013,-39.370,179.630,5.470,149.069
C01712=1208.854,-69.263,-39.358,179.627,5.470,149.070
C01713=1208.859,-69.513,-39.347,179.625,5.470,149.071
C01714=1208.865,-69.763,-39.336,179.622,5.470,149.071
C01715=1208.870,-70.012,-39.325,179.620,5.470,149.072
C01716=1208.875,-70.262,-39.313,179.618,5.470,149.073
C01717=1208.880,-70.512,-39.301,179.616,5.470,149.073
C01718=1208.886,-70.761,-39.291,179.613,5.469,149.074
C01719=1208.891,-71.011,-39.279,179.611,5.469,149.075
C01720=1208.896,-71.261,-39.268,179.609,5.469,149.075
C01721=1208.901,-71.511,-39.257,179.606,5.469,149.076
C01722=1208.907,-71.760,-39.245,179.604,5.469,149.077
C01723=1208.912,-72.010,-39.235,179.602,5.468,149.077
C01724=1208.917,-72.260,-39.223,179.599,5.468,149.078
C01725=1208.922,-72.510,-39.211,179.597,5.468,149.079
C01726=1208.927,-72.759,-39.201,179.594,5.468,149.079
C01727=1208.933,-73.009,-39.189,179.592,5.468,149.080
C01728=1208.938,-73.259,-39.178,179.590,5.468,149.081
C01729=1208.943,-73.508,-39.167,179.587,5.468,149.081
C01730=1208.949,-73.758,-39.156,179.585,5.467,149.082
C01731=1208.953,-74.008,-39.145,179.583,5.467,149.083
C01732=1208.959,-74.257,-39.134,179.581,5.467,149.083
C01733=1208.964,-74.507,-39.123,179.578,5.467,149.084
C01734=1208.969,-74.777,-39.110,179.576,5.467,149.085
C01735=1208.975,-75.048,-39.098,179.573,5.466,149.085
C01736=1208.981,-75.319,-39.086,179.570,5.466,149.086
C01737=1208.986,-75.590,-39.074,179.568,5.466,149.087
C01738=1208.992,-75.839,-39.064,179.566,5.466,149.088
C01739=1208.997,-76.089,-39.052,179.563,5.466,149.088
C01740=1209.002,-76.339,-39.040,179.561,5.466,149.089
C01741=1209.008,-76.588,-39.030,179.558,5.465,149.090
C01742=1209.012,-76.838,-39.019,179.556,5.466,149.090
C01743=1209.018,-77.088,-39.007,179.554,5.465,149.091
C01744=1209.023,-77.337,-38.997,179.551,5.465,149.092
C01745=1209.028,-77.587,-38.986,179.549,5.465,149.092
C01746=1209.033,-77.837,-38.975,179.547,5.464,149.093
C01747=1209.039,-78.086,-38.963,179.544,5.465,149.094
C01748=1209.044,-78.336,-38.952,179.542,5.464,149.094
C01749=1209.049,-78.586,-38.942,179.540,5.464,149.095
C01750=1209.054,-78.835,-38.931,179.537,5.464,149.096
C01751=1209.059,-79.085,-38.920,179.535,5.464,149.096
C01752=1209.065,-79.335,-38.909,179.533,5.464,149.097
C01753=1209.070,-79.585,-38.898,179.530,5.463,149.098
C01754=1209.075,-79.835,-38.887,179.528,5.464,149.098
C01755=1209.080,-80.083,-38.876,179.525,5.463,149.099
C01756=1209.085,-80.334,-38.865,179.524,5.463,149.100
C01757=1209.091,-80.583,-38.854,179.521,5.463,149.100
C01758=1209.096,-80.833,-38.843,179.519,5.463,149.101
C01759=1209.101,-81.083,-38.832,179.516,5.463,149.102
C01760=1209.106,-81.332,-38.822,179.514,5.463,149.102
C01761=1209.111,-81.582,-38.810,179.512,5.463,149.103
C01762=1209.117,-81.832,-38.800,179.509,5.462,149.104
C01763=1209.122,-82.081,-38.788,179.507,5.462,149.104
C01764=1209.127,-82.332,-38.778,179.505,5.462,149.105
C01765=1209.132,-82.581,-38.767,179.502,5.462,149.106
C01766=1209.137,-82.831,-38.756,179.500,5.462,149.107
C01767=1209.143,-83.080,-38.746,179.498,5.462,149.107
C01768=1209.148,-83.330,-38.735,179.496,5.461,149.108
C01769=1209.154,-83.580,-38.724,179.493,5.462,149.108
C01770=1209.159,-83.830,-38.713,179.491,5.461,149.109
C01771=1209.164,-84.080,-38.702,179.488,5.461,149.110
C01772=1209.169,-84.329,-38.691,179.486,5.461,149.111
C01773=1209.174,-84.579,-38.681,179.484,5.460,149.111
C01774=1209.180,-84.829,-38.670,179.482,5.461,149.112
C01775=1209.184,-85.078,-38.659,179.479,5.460,149.112
C01776=1209.190,-85.328,-38.649,179.477,5.461,149.113
C01777=1209.195,-85.577,-38.638,179.474,5.460,149.114
C01778=1209.200,-85.827,-38.627,179.472,5.461,149.115
C01779=1209.206,-86.077,-38.616,179.470,5.460,149.115
C01780=1209.211,-86.327,-38.605,179.468,5.460,149.116
C01781=1209.216,-86.577,-38.595,179.465,5.460,149.116
C01782=1209.221,-86.827,-38.584,179.463,5.459,149.117
C01783=1209.226,-87.076,-38.573,179.461,5.460,149.118
C01784=1209.231,-87.326,-38.563,179.458,5.459,149.119
C01785=1209.237,-87.576,-38.552,179.456,5.459,149.119
C01786=1209.242,-87.825,-38.541,179.454,5.459,149.120
C01787=1209.247,-88.075,-38.531,179.451,5.459,149.121
C01788=1209.252,-88.325,-38.520,179.449,5.459,149.121
C01789=1209.258,-88.574,-38.509,179.447,5.459,149.122
C01790=1209.263,-88.824,-38.499,179.445,5.458,149.122
C01791=1209.268,-89.074,-38.489,179.442,5.459,149.123
C01792=1209.273,-89.323,-38.477,179.440,5.458,149.124
C01793=1209.279,-89.573,-38.467,179.438,5.459,149.125
C01794=1209.284,-89.823,-38.456,179.435,5.458,149.125
C01795=1209.289,-90.073,-38.446,179.433,5.458,149.126
C01796=1209.294,-90.322,-38.435,179.431,5.458,149.126
C01797=1209.299,-90.572,-38.425,179.428,5.457,149.127
C01798=1209.304,-90.822,-38.414,179.426,5.458,149.128
C01799=1209.310,-91.072,-38.404,179.423,5.457,149.129
C01800=1209.315,-91.321,-38.393,179.421,5.458,149.129
C01801=1209.320,-91.571,-38.383,179.419,5.457,149.130
C01802=1209.326,-91.820,-38.372,179.417,5.457,149.131
C01803=1209.331,-92.071,-38.362,179.414,5.457,149.131
C01804=1209.336,-92.320,-38.352,179.412,5.457,149.132
C01805=1209.341,-92.570,-38.340,179.410,5.457,149.133
C01806=1209.347,-92.819,-38.330,179.408,5.457,149.133
C01807=1209.352,-93.069,-38.319,179.405,5.456,149.134
C01808=1209.357,-93.319,-38.309,179.403,5.457,149.135
C01809=1209.362,-93.569,-38.299,179.400,5.456,149.135
C01810=1209.368,-93.819,-38.288,179.398,5.457,149.136
C01811=1209.373,-94.067,-38.278,179.396,5.456,149.136
C01812=1209.378,-94.318,-38.268,179.394,5.456,149.137
C01813=1209.383,-94.567,-38.257,179.391,5.456,149.138
C01814=1209.388,-94.817,-38.247,179.389,5.456,149.139
C01815=1209.394,-95.067,-38.237,179.387,5.456,149.139
C01816=1209.399,-95.317,-38.226,179.385,5.456,149.140
C01817=1209.404,-95.567,-38.216,179.382,5.455,149.140
C01818=1209.410,-95.816,-38.206,179.380,5.455,149.141
C01819=1209.415,-96.066,-38.194,179.378,5.455,149.142
C01820=1209.420,-96.316,-38.184,179.375,5.455,149.143
C01821=1209.424,-96.565,-38.174,179.373,5.455,149.143
C01822=1209.430,-96.815,-38.164,179.371,5.454,149.144
